# B&R Automation Studio project EFI (part 22)

#### OutputsP5.st
```iecst
ACTION OutputsP5:

(*CABINET 01*)

	//X20DOF322_009
	X20DOF322_009.DOutput[1]:=gBlockOutputs[1].xShotLine1;
	X20DOF322_009.DOutput[2]:=gBlockOutputs[1].xShotLine2;
	X20DOF322_009.DOutput[3]:=gBlockOutputs[1].xEnableDobleShot;
	X20DOF322_009.DOutput[4]:=gMachine.Out.xResetCB1;
	X20DOF322_009.DOutput[5]:=gMachine.Out.xResetRouter;
	X20DOF322_009.DOutput[6]:= FALSE;								//SPARE
	X20DOF322_009.DOutput[7]:=gMachine.Out.xAirSupply;
	X20DOF322_009.DOutput[8]:=gMachine.Out.xGreenLight;
	X20DOF322_009.DOutput[9]:=gMachine.Out.xLightReset;
	X20DOF322_009.DOutput[10]:=gMachine.Out.xBuzzerButtonPanel;
	X20DOF322_009.DOutput[11]:= TRUE;
	X20DOF322_009.DOutput[12]:= FALSE;								//SPARE
	X20DOF322_009.DOutput[13]:= FALSE;								//SPARE
	X20DOF322_009.DOutput[14]:= FALSE;								//SPARE
	X20DOF322_009.DOutput[15]:= FALSE;								//SPARE
	X20DOF322_009.DOutput[16]:= FALSE;								//SPARE

	// X20DOF322_010
	X20DOF322_010.DOutput[1]:= gInksOutputs[1].xOutPowPrintHead;
	X20DOF322_010.DOutput[2]:= gInksOutputs[2].xOutPowPrintHead;
	X20DOF322_010.DOutput[3]:= gInksOutputs[3].xOutPowPrintHead;
	X20DOF322_010.DOutput[4]:= gInksOutputs[4].xOutPowPrintHead;
	X20DOF322_010.DOutput[5]:= gInksOutputs[5].xOutPowPrintHead;
	X20DOF322_010.DOutput[6]:= gInksOutputs[6].xOutPowPrintHead;
	X20DOF322_010.DOutput[7]:= gInksOutputs[7].xOutPowPrintHead;
	X20DOF322_010.DOutput[8]:= gInksOutputs[8].xOutPowPrintHead;
	X20DOF322_010.DOutput[9]:= gInksOutputs[1].xOutBarResistance;
	X20DOF322_010.DOutput[10]:= gInksOutputs[2].xOutBarResistance;
	X20DOF322_010.DOutput[11]:= gInksOutputs[3].xOutBarResistance;
	X20DOF322_010.DOutput[12]:= gInksOutputs[4].xOutBarResistance;
	X20DOF322_010.DOutput[13]:= gInksOutputs[5].xOutBarResistance;
	X20DOF322_010.DOutput[14]:= gInksOutputs[6].xOutBarResistance;
	X20DOF322_010.DOutput[15]:= gInksOutputs[7].xOutBarResistance;
	X20DOF322_010.DOutput[16]:= gInksOutputs[8].xOutBarResistance;

	//X20DOF322_011
	X20DOF322_011.DOutput[1] := gInksOutputs[1].xSolenoid1;
	X20DOF322_011.DOutput[2] := gInksOutputs[2].xSolenoid1;
	X20DOF322_011.DOutput[3] := gInksOutputs[1].xSolenoid2;
	X20DOF322_011.DOutput[4] := gInksOutputs[2].xSolenoid2;
	X20DOF322_011.DOutput[5] := gInksOutputs[3].xSolenoid1;
	X20DOF322_011.DOutput[6] := gInksOutputs[4].xSolenoid1;
	X20DOF322_011.DOutput[7] := gInksOutputs[3].xSolenoid2;
	X20DOF322_011.DOutput[8] := gInksOutputs[4].xSolenoid2;
	X20DOF322_011.DOutput[9] := gInksOutputs[5].xSolenoid1;
	X20DOF322_011.DOutput[10] := gInksOutputs[6].xSolenoid1;
	X20DOF322_011.DOutput[11] := gInksOutputs[5].xSolenoid2;
	X20DOF322_011.DOutput[12] := gInksOutputs[6].xSolenoid2;
	X20DOF322_011.DOutput[13] := gInksOutputs[7].xSolenoid1;
	X20DOF322_011.DOutput[14] := gInksOutputs[8].xSolenoid1;
	X20DOF322_011.DOutput[15] := gInksOutputs[7].xSolenoid2;
	X20DOF322_011.DOutput[16] := gInksOutputs[8].xSolenoid2;

	//X20DOF322_012
	X20DOF322_012.DOutput[1]:=gInksOutputs[1].xReliefValve;
	X20DOF322_012.DOutput[2]:=gInksOutputs[2].xReliefValve;
	X20DOF322_012.DOutput[3]:=gInksOutputs[3].xReliefValve;
	X20DOF322_012.DOutput[4]:=gInksOutputs[4].xReliefValve;
	X20DOF322_012.DOutput[5]:=gInksOutputs[5].xReliefValve;
	X20DOF322_012.DOutput[6]:=gInksOutputs[6].xReliefValve;
	X20DOF322_012.DOutput[7]:=gInksOutputs[7].xReliefValve;
	X20DOF322_012.DOutput[8]:=gInksOutputs[8].xReliefValve;
	X20DOF322_012.DOutput[9]:= FALSE;								//SPARE
	X20DOF322_012.DOutput[10]:=FALSE;								//SPARE
	X20DOF322_012.DOutput[11]:=FALSE;								//SPARE
	X20DOF322_012.DOutput[12]:=FALSE;								//SPARE
	X20DOF322_012.DOutput[13]:=FALSE;								//SPARE
	X20DOF322_012.DOutput[14]:=FALSE;								//SPARE
	X20DOF322_012.DOutput[15]:=FALSE;								//SPARE
	X20DOF322_012.DOutput[16]:=FALSE;								//SPARE

	//X20DOF322_013
	X20DOF322_013.DOutput[1]:=gMachine.Out.xConsentL1;
	X20DOF322_013.DOutput[2]:=gMachine.Out.xConsentL2;
	X20DOF322_013.DOutput[3]:=gMachine.Out.xCompenserLine1;
	X20DOF322_013.DOutput[4]:=gMachine.Out.xCompenserLine2;
	X20DOF322_013.DOutput[5]:=gMachine.Out.xYellowLight;
	X20DOF322_013.DOutput[6]:=gMachine.Out.xRedLight;
	X20DOF322_013.DOutput[7]:=gMachine.Out.xLine1ReadyToClean;
	X20DOF322_013.DOutput[8]:=gMachine.Out.xLine2ReadyToClean;
	X20DOF322_013.DOutput[9]:=gMachine.Out.xSuctionTurbine;
	X20DOF322_013.DOutput[10]:= gJamDetect[1].Outputs.xJamTestSignal[1] OR gJamDetect[2].Outputs.xJamTestSignal[1];
	X20DOF322_013.DOutput[11]:=gJamDetect[1].Outputs.xJamTestSignal[2] OR gJamDetect[2].Outputs.xJamTestSignal[2];
	X20DOF322_013.DOutput[12]:=gJamDetect[1].Outputs.xJamTestSignal[3] OR gJamDetect[2].Outputs.xJamTestSignal[3];
	X20DOF322_013.DOutput[13]:=gJamDetect[1].Outputs.xJamTestSignal[4] OR gJamDetect[2].Outputs.xJamTestSignal[4];
	X20DOF322_013.DOutput[14]:= FALSE;								//SPARE
	X20DOF322_013.DOutput[15]:= FALSE;								//SPARE
	X20DOF322_013.DOutput[16]:= FALSE;								//SPARE

	// X20AO4622_017 	(*  BAR A *) 	(*  BAR B *)
	X20AO4622_017.AOutput[1]:= gInksOutputs[1].iDutyCycleNegative;
	X20AO4622_017.AOutput[2]:= gInksOutputs[2].iDutyCycleNegative;
	X20AO4622_017.AOutput[3]:= gInksOutputs[1].iDutyCycleFilling;
	X20AO4622_017.AOutput[4]:= gInksOutputs[2].iDutyCycleFilling;

	// X20AO4622_018 	(*  BAR C *) 	(*  BAR D *)
	X20AO4622_018.AOutput[1]:= gInksOutputs[3].iDutyCycleNegative;
	X20AO4622_018.AOutput[2]:= gInksOutputs[4].iDutyCycleNegative;
	X20AO4622_018.AOutput[3]:= gInksOutputs[3].iDutyCycleFilling;
	X20AO4622_018.AOutput[4]:= gInksOutputs[4].iDutyCycleFilling;

	// X20AO4622_019 	(*  BAR E *) 	(*  BAR F *)
	X20AO4622_019.AOutput[1]:= gInksOutputs[5].iDutyCycleNegative;
	X20AO4622_019.AOutput[2]:= gInksOutputs[6].iDutyCycleNegative;
	X20AO4622_019.AOutput[3]:= gInksOutputs[5].iDutyCycleFilling;
	X20AO4622_019.AOutput[4]:= gInksOutputs[6].iDutyCycleFilling;

	// X20AO4622_020 	(*  BAR G *) 	(*  BAR H *)
	X20AO4622_020.AOutput[1]:= gInksOutputs[7].iDutyCycleNegative;
	X20AO4622_020.AOutput[2]:= gInksOutputs[8].iDutyCycleNegative;
	X20AO4622_020.AOutput[3]:= gInksOutputs[7].iDutyCycleFilling;
	X20AO4622_020.AOutput[4]:= gInksOutputs[8].iDutyCycleFilling;

	// X20AO4622_100 THICKNESS SENSOR RESET
	X20AI2636_100.DOutput[1] := gDing.Out.xReset;;  // Reset the target fault

	// SI UNIT BK1
	SiUnitPwrLnkBK1.Output01_16.0 := gBlockOutputs[1].xTrayIn;
	SiUnitPwrLnkBK1.Output01_16.1 := gBlockOutputs[1].xTrayOut;
	SiUnitPwrLnkBK1.Output01_16.2 := gMachine.commands.CleanBelt.xCleanBeltPump;
	SiUnitPwrLnkBK1.Output01_16.3 := gBlockOutputs[1].xVenturi;
	SiUnitPwrLnkBK1.Output01_16.4 := gBlockOutputs[1].xCleaningWaterPump;
	SiUnitPwrLnkBK1.Output01_16.5 := gMachine.commands.CleanBelt.xPistonFlojet;
	SiUnitPwrLnkBK1.Output01_16.6 := FALSE;
	SiUnitPwrLnkBK1.Output01_16.7 := FALSE;
	SiUnitPwrLnkBK1.Output01_16.8 := FALSE;
	SiUnitPwrLnkBK1.Output01_16.9 := FALSE;
	SiUnitPwrLnkBK1.Output01_16.10 := FALSE;
	SiUnitPwrLnkBK1.Output01_16.11 := FALSE;
	SiUnitPwrLnkBK1.Output01_16.12 := FALSE;
	SiUnitPwrLnkBK1.Output01_16.13 := FALSE;
	SiUnitPwrLnkBK1.Output01_16.14 := FALSE;
	SiUnitPwrLnkBK1.Output01_16.15 := FALSE;

END_ACTION
```

#### OutputsShield.st
```iecst
ACTION OutputsShield:

	//X3 PLC
	X3.DOutput[1]:= FALSE;
	X3.DOutput[2]:= gMachine.Out.xPC2Start;
	X3.DOutput[3]:= gMachine.Out.xResetCB1;
	X3.DOutput[4]:= gMachine.Out.xResetRouter;

	// X20DOF322_005
	X20DOF322_005.DOutput[1]	:= gInksOutputs[1].xOutPowPrintHead;
	X20DOF322_005.DOutput[2]	:= gInksOutputs[2].xOutPowPrintHead;
	X20DOF322_005.DOutput[3]	:= gInksOutputs[1].xOutBarResistance;
	X20DOF322_005.DOutput[4]	:= gInksOutputs[2].xOutBarResistance;
	X20DOF322_005.DOutput[5]	:= gInksOutputs[1].xSolenoid1;
	X20DOF322_005.DOutput[6]	:= gInksOutputs[2].xSolenoid1;
	X20DOF322_005.DOutput[7]	:= gInksOutputs[1].xSolenoid2;
	X20DOF322_005.DOutput[8]	:= gInksOutputs[2].xSolenoid2;
	X20DOF322_005.DOutput[9]	:= gInksOutputs[1].xReliefValve;
	X20DOF322_005.DOutput[10]	:= gInksOutputs[2].xReliefValve;
	X20DOF322_005.DOutput[11]	:= FALSE;
	X20DOF322_005.DOutput[12]	:= gChiller[1].Out.xStart;
	X20DOF322_005.DOutput[13]	:= gMachine.Out.xCoolingPCStart;//Implement
	X20DOF322_005.DOutput[14]	:= gBlock[1].Out.xEnableDobleShot;
	X20DOF322_005.DOutput[15]	:= gBlock[1].Out.xShotLine1;
	X20DOF322_005.DOutput[16]	:= gBlock[1].Out.xShotLine2;

	// X20DOF322_006
	X20DOF322_006.DOutput[1]	:= gMachine.Out.xConsentL1;
	X20DOF322_006.DOutput[2]	:= gMachine.Out.xConsentL2;
	X20DOF322_006.DOutput[3]	:= gMachine.Out.xCompenserLine1;
	X20DOF322_006.DOutput[4]	:= gMachine.Out.xCompenserLine2;
	X20DOF322_006.DOutput[5]	:= gMachine.Out.xYellowLight;
	X20DOF322_006.DOutput[6]	:= gMachine.Out.xRedLight;
	X20DOF322_006.DOutput[7]	:= gMachine.Out.xLine1ReadyToClean;
	X20DOF322_006.DOutput[8]	:= gMachine.Out.xLine2ReadyToClean;
	X20DOF322_006.DOutput[9]	:= gMachine.Out.xSuctionTurbine;
	X20DOF322_006.DOutput[10]	:= FALSE;
	X20DOF322_006.DOutput[11]	:= FALSE;
	X20DOF322_006.DOutput[12]	:= TRUE;
	X20DOF322_006.DOutput[13]	:= gMachine.Out.xAirSupply;
	X20DOF322_006.DOutput[14]	:= gMachine.Out.xGreenLight;
	X20DOF322_006.DOutput[15]	:= gMachine.Out.xLightReset;
	X20DOF322_006.DOutput[16]	:= gMachine.Out.xBuzzerButtonPanel;

	// SI UNIT BK1
	SiUnitBK1.Output01_08.0		:= gBlockOutputs[1].xTrayIn;
	SiUnitBK1.Output01_08.1		:= gBlockOutputs[1].xTrayOut;
	SiUnitBK1.Output01_08.2		:= gMachine.commands.CleanBelt.xCleanBeltPump;
	SiUnitBK1.Output01_08.3		:= gBlockOutputs[1].xVenturi;
	SiUnitBK1.Output01_08.4		:= gMachine.commands.CleanBelt.xPistonFlojet;
	SiUnitBK1.Output01_08.5		:= gBlockOutputs[1].xCleaningWaterPump;

	// X20AO4622_009	 (*  BAR A *)	 (*  BAR B *)
	X20AO4622_009.AOutput[1]:= gInksOutputs[1].iDutyCycleNegative;
	X20AO4622_009.AOutput[2]:= gInksOutputs[2].iDutyCycleNegative;
	X20AO4622_009.AOutput[3]:= gInksOutputs[1].iDutyCycleFilling;
	X20AO4622_009.AOutput[4]:= gInksOutputs[2].iDutyCycleFilling;

END_ACTION
```

### Program Logical/Printer/Sim/SimMachine (IEC)

#### Main.st - Init, cyclic, exit code
```iecst
PROGRAM _INIT

	URLHost := '127.0.0.1';

	Initialization;

	//Call variables to avoid unusefull warnings
	// Simple modification
	GlobalIO;
	DeviceComms;
	Dryer;
	InkBox;
	Motion;

END_PROGRAM

PROGRAM _CYCLIC

	MachineModelCode;

	General;

	UPS;

	Tests;

	LogTests;

	//Definition of the machine at the end of the code
	IF simMachineTypeEnumCopy<>gSimMachine.Parameters.MachineType THEN
		simMachineType := DINT_TO_INT(gSimMachine.Parameters.MachineType);
		IF simMachineTypeEnumCopy <> SIM_MACHINE_REAL THEN
			xNeedToRestartCPU := TRUE;
		END_IF
	END_IF
	IF simMachineType<>simMachineTypeCopy THEN
		gSimMachine.Parameters.MachineType := simMachineType;
	END_IF

	simMachineTypeCopy := simMachineType;
	simMachineTypeEnumCopy := gSimMachine.Parameters.MachineType;

	//Restart CPU if needed. Done with timer to allow other programs to use the new model and save it before restart
	tonRestart.IN := xNeedToRestartCPU;
	tonRestart.PT := T#300ms;
	tonRestart();
	IF tonRestart.Q THEN
		statusReset := SYSreset(enable:= TRUE, mode:= 2);
	END_IF

END_PROGRAM

PROGRAM _EXIT
	gEventLogManager; //Just here to be able to watch this var
END_PROGRAM
```

#### GlobalVariables.st
```iecst
ACTION GlobalIO:
	X20CPUData; (*Map: P4&EBRO*)
	X1; (*Map: P4&EBRO*)
	X2; (*Map: P4&EBRO*)
	X3; (*Map: P4&EBRO*)
	X20DOF322_001; (*Map: P4*)
	X20DIF371_001; (*Map: EBRO&S1400*)
	X20DIF371_002; (*Map: P4&EBRO&S1400*)
	X20DIF371_003; (*Map: P4&EBRO$S1400*)
	X20DOF322_004; (*Map: P4*)
	X20DIF371_004; (*Map: EBRO*)
	X20DIF371_005; (*Map: S1400*)
	X20DIF371_006; (*Map: S1400*)
	X20AI2636_005; (*Map: P4*)
	X20DOF322_005; (*Map: EBRO*)
	X20SLX402_006; (*	X20SI2100_010; Map: P4*)
	X20DOF322_006; (*Map: EBRO*)
	X20AI4322_008; (*Map: EBRO*)
	X20AI4322_102; (*Map: InkBox*)
	X20AI4322_202; (*Map: InkBox*)
	X20AI4322_302; (*Map: InkBox*)
	X20AT2222_103; (*Map: InkBox*)
	X20AT2222_203; (*Map: InkBox*)
	X20AT2222_303; (*Map: InkBox*)
	X20DOF322_104; (*Map: InkBox*)
	X20DOF322_204; (*Map: InkBox*)
	X20DOF322_304; (*Map: InkBox*)
	X20AO4622_105; (*Map: InkBox*)
	X20AO4622_205; (*Map: InkBox*)
	X20AO4622_305; (*Map: InkBox*)
	X20DI9372_008; (*Map: S1400*)
	X20AO4622_009; (*Map: EBRO*)
	X20DOF322_009; (*Map:S1400*)
	X20DOF322_010; (*Map:S1400*)
	X20AT4222_010; (*Map: EBRO*)
	X20DOF322_011; (*Map:S1400*)
	X20DOF322_012; (*Map:S1400*)
	X20DOF322_013; (*Map:S1400*)
	X20AI8321_015; (*Map:S1400*)
	X20AI8321_016; (*Map:S1400*)
	X20AI8321_111; (*Map:S1400*)
	X20AI8321_112; (*Map:S1400*)
	X20AI8321_113; (*Map:S1400*)
	X20AI8321_018; (*Map:S1400*)
	X20AI8321_019; (*Map:S1400*)
	X20AO4622_017; (*Map:S1400*)
	X20AO4622_018; (*Map:S1400*)
	X20AO4622_019; (*Map:S1400*)
	X20AO4622_020; (*Map:S1400*)
	X20AT4222_022; (*Map:S1400*)
	X20AT4222_023; (*Map:S1400*)
	X20AI2636_024; (*Map:S1400*)
	X20AI8321_025;
	X20AI8321_024;
	X20DIF371_024; (*Map:S1400*)
	X20AI8321_026; (*Map:S1400*)
	X20AT4222_027;
	X20AT4222_028;
	X20AT4222_029; (*Map:S1400*)
	X20AT4222_030; (*Map:S1400*)
	X20DIF371_030; (*Map: P4*)
	X20AI2636_100;
	X20DIF371_101; (*Map: P4 & Map: InkBox*)
	X20DIF371_102; (*Map: P4*)
	X20DIF371_103; (*Map: P4*)
	X20DIF371_104; (*Map: P4*)
	X20DIF371_105; (*Map: P4*)
	X20DIF371_106; (*Map: P4*)
	X20DI9372_107; (*Map: P4*)
	X20DIF371_107; (*Map: P4*)
	X20DC4395_104; (*Map: P4*)
	X20DC4395_105; (*Map: P4*)
	X20DOF322_106; (*Map: P4*)
	X20DOF322_107; (*Map: P4*)
	X20DOF322_108; (*Map: P4*)
	X20DOF322_109; (*Map: P4*)
	X20DOF322_110; (*Map: P4*)
	X20AI8321_109; (*Map: P4*)
	X20AI8321_110; (*Map: P4*)
	X20AO4622_111; (*Map: P4*)
	X20AO4622_112; (*Map: P4*)
	X20AO4622_113; (*Map: P4*)
	X20AO4622_114; (*Map: P4*)
	X20AO4622_115; (*Map: P4*)
	X20AO4622_116; (*Map: P4*)
	X20AO4622_117; (*Map: P4*)
	X20AT4222_114; (*Map: P4*)
	X20AT4222_115; (*Map: P4*)
	X20AT4222_116; (*Map: P4*)
	X20AT4222_117; (*Map: P4*)
	X20AT4222_118; (*Map: P4*)
	X20AT4222_119; (*Map: P4*)
	X20AT4222_120; (*Map: P4*)
	X20AT4222_121; (*Map: P4*)
	X20CS1030_150; (*Map: P4*)
	X20CS1030_151; (*Map: P4*)
	X20PS3300_114; (*Map: P4*)
	X20PS3300_106; (*Map: P4*)
	X20PS3300_152; (*Map: P4*)
	X20DIF371_153; (*Map: P4*)
	X20DIF371_154; (*Map: P4*)
	X20DOF322_155; (*Map: P4*)
	X20AI8221_156; (*Map: P4*)
	X20AO4622_157; (*Map: P4*)
	X20AO4622_158; (*Map: P4*)
	X20SI8110_117; (*Map: P4*)
	X20SO2110_118; (*Map: P4*)
	X20DIF371_201; (*Map: P4 & InkBox*)
	X20DIF371_202; (*Map: P4*)
	X20DIF371_203; (*Map: P4*)
	X20DIF371_301; (*Map: InkBox*)
	X20DC4395_204; (*Map: P4*)
	X20DC4395_205; (*Map: P4*)
	X20DOF322_205; (*Map: Dryer*)
	X20DOF322_206; (*Map: P4*)
	X20DOF322_207; (*Map: P4*)
	X20DOF322_208; (*Map: P4*)
	X20AI8321_207; (*Map: P4*)
	X20AI8321_209; (*Map: P4*)
	X20AI8321_210; (*Map: P4*)
	X20AO4622_208; (*Map: Dryer*)
	X20AO4622_211; (*Map: P4*)
	X20AO4622_212; (*Map: P4*)
	X20AO4622_213; (*Map: P4*)
	X20AT4222_209; (*Map: Dryer*)
	X20AT4222_214; (*Map: P4*)
	X20AT4222_215; (*Map: P4*)
	X20AT4222_216; (*Map: P4*)
	X20SI8110_217; (*Map: P4*)
	X20SO2110_218; (*Map: P4*)
	Reserve01;
	SiUnitBK1;
	SiUnitBK2;
	SiUnitPwrLnkBK1;
	Pdc_X20DIF371_001;
	Pdc_X20DIF371_002;
	Pdc_X20DIF371_003;
	Pdc_X20DIF371_004;
	Pdc_X20DIF371_005;
	Pdc_X20DIF371_006;
	X20PS3300_007;
	Pdc_X20DIF371_020;
	Pdc_X20DIF371_021;
	X20PS3300_022;
	Pdc_X20DOF322_023;
	Pdc_X20DIF371_1;
	Pdc_X20DIF371_2;
	Pdc_X20DIF371_3;
	Pdc_X20DOF322_008;
	Pdc_X20DOF322_009;
	Pdc_X20DOF322_010;
	Pdc_X20DOF322_1;
	Pdc_X20DIF371_040;
	Pdc_X20DOF322_011;
	X20IF1072_SS1;
	X20SM1436_007;
	X20SM1436_008;
	X20SM1436_011;
	X20SM1436_012;
	X20SM1436_111;
	X20SM1436_112;
	X20PS3300_014;
	X20PS3300_021;
	X20BC0083;
	X20PS9400;
END_ACTION

ACTION DeviceComms:
	gIclaNetData;

	gReceivedDataModbTransport;
	gToWriteDataModbTransport;

END_ACTION

ACTION Dryer:

	gDryer;
	gDryerLocalData;
	gDryerRemoteData;
	gNirAdphos;
	gArcLampGew;
	gSimpleBlock;
	gIndexSimpleBlock;

	gPermanentArcLampGew;
	gPermanentNirAdphos;
	gPermanentDryer;
	gPermanentInkBox;
	gPermanentSimpleBlock;

	gSimArcLamp;
	gSimNirAdphos;
	gSimSimpleBlock;

END_ACTION

ACTION InkBox:

	gInkBox;

END_ACTION

ACTION Motion:

	gAxisStepper;

END_ACTION
```

#### SimMachine.var - Local variables
```iecst
VAR
	iIndexPsu : USINT;
	iSimIndex : USINT; (*Index for loops in simulation*)
	simEventLog : EventLog_typ;
	webClient : httpClient;
	ResponseHeader : httpResponseHeader_t;
	RequestData : STRING[3000];
	ResponseData : STRING[3000];
	URLHost : STRING[80];
	URIHost : STRING[80];
	xTestPrepareMachine : BOOL; (*This value must be used as active while pressed by the visualization*)
	xTestPrePrepare : BOOL; (*This value must be used as active while pressed by the visualization*)
	xTestBeltTests : BOOL; (*This value must be used as active while pressed by the visualization*)
	xTestConsents : BOOL; (*This value must be used as active while pressed by the visualization*)
	xTestBlock : BOOL; (*This value must be used as active while pressed by the visualization*)
	xTestTrVacuum : BOOL;
	xTestLine : BOOL; (*This value must be used as active while pressed by the visualization*)
	xTestCleaning : BOOL; (*This value must be used as active while pressed by the visualization*)
	testMonitor : UtMgrMonitor;
	ctrlBlock2 : UINT;
	simMachineType : INT;
	simMachineTypeCopy : INT;
	simMachineTypeEnumCopy : SimMachineType;
	xBlockExists2 : BOOL;
	statusReset : UINT;
	tonRestart : TON;
	xNeedToRestartCPU : BOOL;
	stEventLogTests : EventLog_typ;
END_VAR
```

### Program Logical/Printer/Sim/SimMachine_Fast (IEC)

#### Main.st - Init, cyclic, exit code
```iecst
PROGRAM _INIT

	InitialDataForMedia;
	PreparingMethodComms;

	InitialDataForMediaEnergy;
	PreparingMethodEnergyComms;

END_PROGRAM

PROGRAM _CYCLIC

	Media;

	// Sending information to the new boards
	Stack;
	StackEnergy;

END_PROGRAM
```

#### StackEnergy.st
```iecst
ACTION StackEnergy:

	(* UA_MethodCall - call methode *)
	InputArguments_Energy[0].Name := 'MediaData';
	InputArguments_Energy[0].Value := '::SimMachFst:NewMediaData_Energy';
	OutputArguments_Energy[0].Name := 'Result';
	OutputArguments_Energy[0].Value := '::SimMachFst:MethodResult_Energy';
	UA_MethodCall_Energy(Execute := ExecuteMethodCall_Energy,
		ConnectionHdl := ConnectionHdl_Energy,
		MethodHdl := MethodHdl_Energy,
		Timeout := T#10s,
		InputArguments := InputArguments_Energy,
		OutputArguments := OutputArguments_Energy);
	IF NOT UA_MethodCall_Energy.Busy THEN
		ExecuteMethodCall_Energy := FALSE;
		IF UA_MethodCall_Energy.Done THEN
			NewMediaData_Energy.MediaData.rLength := NewMediaData_Energy.MediaData.rLength + 1;
		END_IF
		IF UA_MethodCall_Energy.Error THEN
			NewMediaData_Energy.MediaData.rDocLength := NewMediaData_Energy.MediaData.rDocLength + 1;
		END_IF
	END_IF

	// Managing the automatic sending. Just Energy when enabled to Dry
	IF NOT gThicknessCtrl.status.xNewMediaStackEnabled OR NOT gThicknessCtrl.parameters.Dry.xDryStack THEN
		RETURN;
	END_IF

	IF (gSimMachine.Parameters.Stack.iMediaQuantityToKeepLoaded <= gThicknessCtrl.status.Stack.iNewMediaLoadedL1 + gThicknessCtrl.status.Stack.iNewMediaLoadedL2) THEN
		RETURN;
	END_IF

	// Adding a timer to avoid not working the method
	tonNotCallingMethod_Energy.IN := NOT UA_MethodCall_Energy.Busy;
	tonNotCallingMethod_Energy.PT := t#500ms;
	tonNotCallingMethod_Energy();
	IF EDGEPOS(tonNotCallingMethod_Energy.Q) THEN
		ExecuteMethodCall_Energy := TRUE;
	END_IF

END_ACTION

ACTION InitialDataForMediaEnergy:

	NewMediaData_Energy.MediaData.iLine := 1;
	NewMediaData_Energy.MediaData.xHasWhite := FALSE;
	NewMediaData_Energy.MediaData.rThickness := 3;
	NewMediaData_Energy.MediaData.rMargin := 2;
	NewMediaData_Energy.MediaData.rWidth := 1400;
	NewMediaData_Energy.MediaData.rLength := 1000;
	NewMediaData_Energy.MediaData.rCrossOffset := -700;
	NewMediaData_Energy.MediaData.rDocWidth := 1400;
	NewMediaData_Energy.MediaData.rDocLength := 950;
	NewMediaData_Energy.MediaData.rDocCrossOffset := -700;
	NewMediaData_Energy.MediaData.rDocProcessOffset := 0;

	//Just to see some data
	NewMediaData_Energy.Energy.iPower[0,0] := 50;
	NewMediaData_Energy.Energy.iPower[1,0] := 50;
	NewMediaData_Energy.Energy.iPower[0,1] := 50;

END_ACTION

ACTION PreparingMethodEnergyComms:

	ExecuteConnect_Energy := TRUE;

	(* UA_Connect - establish connection to OPC UA Server *)
	SessionConnectInfo_Energy.SecurityMsgMode := UASecurityMsgMode_None;
	SessionConnectInfo_Energy.SecurityPolicy := UASecurityPolicy_None;
	SessionConnectInfo_Energy.TransportProfile := UATP_UATcp;
	SessionConnectInfo_Energy.UserIdentityToken.UserIdentityTokenType := UAUITT_Username;
	SessionConnectInfo_Energy.UserIdentityToken.TokenParam1 := 'PressCore';
	SessionConnectInfo_Energy.UserIdentityToken.TokenParam2 := 'h98o76';
	SessionConnectInfo_Energy.SessionTimeout := T#1m;
	SessionConnectInfo_Energy.MonitorConnection := T#10s;

	UA_Connect_Energy(Execute := ExecuteConnect_Energy,
		ServerEndpointUrl := 'opc.tcp://localhost:4840',
		SessionConnectInfo := SessionConnectInfo_Energy,
		Timeout := T#10s);
	IF NOT UA_Connect_Energy.Busy THEN
		ExecuteConnect_Energy := FALSE;
		IF UA_Connect_Energy.Done THEN
			ConnectionHdl_Energy := UA_Connect_Energy.ConnectionHdl;
			////// NEXT
			ExecuteGetnamespaceindex_Energy := TRUE;
		END_IF
		IF UA_Connect_Energy.Error THEN
			ConnectionHdl_Energy := 0;
		END_IF
	END_IF

	(* UA_GetNamespaceIndex - read index of required namespace for PVs *)
	UA_GetNamespaceIndex_Energy(Execute := ExecuteGetnamespaceindex_Energy,
		ConnectionHdl := ConnectionHdl_Energy,
		NamespaceUri := 'http://br-automation.com/OpcUa/PLC/PV/',
	Timeout := T#5s);
	IF NOT UA_GetNamespaceIndex_Energy.Busy THEN
		ExecuteGetnamespaceindex_Energy := FALSE;
		IF UA_GetNamespaceIndex_Energy.Done THEN
			NamespaceIndex_Energy := UA_GetNamespaceIndex_Energy.NamespaceIndex;
			////// NEXT
			ExecuteMethodGetHandle_Energy := TRUE;
		END_IF
		IF UA_GetNamespaceIndex_Energy.Error THEN
			NamespaceIndex_Energy := 0;
		END_IF
	END_IF

	(* UA_MethodGetHandle - get a handle for required methode *)
	ObjectNodeID_Energy.NamespaceIndex := NamespaceIndex_Energy;
	ObjectNodeID_Energy.Identifier := '::ThickPos';
	ObjectNodeID_Energy.IdentifierType := UAIdentifierType_String;
	MethodNodeID_Energy.NamespaceIndex := NamespaceIndex_Energy;
	MethodNodeID_Energy.Identifier := '::ThickPos:LoadNewMediaEnergy';
	MethodNodeID_Energy.IdentifierType := UAIdentifierType_String;
	UA_MethodGetHandle_Energy(Execute := ExecuteMethodGetHandle_Energy,
		ConnectionHdl := ConnectionHdl_Energy,
		ObjectNodeID := ObjectNodeID_Energy,
		MethodNodeID := MethodNodeID_Energy,
		Timeout := T#10s);
	IF NOT UA_MethodGetHandle_Energy.Busy THEN
		ExecuteMethodGetHandle_Energy := FALSE;
		IF UA_MethodGetHandle_Energy.Done THEN
			MethodHdl_Energy := UA_MethodGetHandle_Energy.MethodHdl;
			////// NEXT
			// READY TO COMMUNICATE
		END_IF
		IF UA_MethodGetHandle_Energy.Error THEN
			MethodHdl_Energy := 0;
		END_IF
	END_IF

END_ACTION
```

- Visualisation Logical/Printer/Sim/SimVisu (not shown)

### Program Logical/Printer/Sim/TestResources (IEC)

#### TestResources.st - Init, cyclic, exit code
```iecst
PROGRAM _CYCLIC

	rVal := 0.6; //Complex value. Just a starting value
	FOR iIndex:=0 TO iMax DO
		rVal := rVal * SQRT(rVal);
	END_FOR;

END_PROGRAM
```

- Remote&LocalParams.graphml (not shown)

### Package Logical/Dryer/Config - Machine configurator

### Program Logical/Dryer/Config/Initialize (IEC) - Initialize program

#### Initialize.var
```iecst
VAR
	HWInfoCpu : HWInfo;
	projectInfo : ArProjectGetInfo;
END_VAR
```

### Program Logical/Dryer/Config/MachineConfigurator (IEC) - Machine configurator

#### MachineModel.st - Constant values according machine model
```iecst
ACTION MachineModel:

	//Assignation of machine model just when unnasigned
	IF gDryer.In.iMachineModelCode=0 THEN
		InputsMachineModel;
	END_IF

	// MachineModelAssignation
	// From the inputs of the type of machine readed by the inputs to the Parameter of the particular Type of Machine
	CASE gDryer.Pt.ConfigNameID OF

		GC_CONFIG_DRYER_NOZ2_ID:
			CASE gDryer.In.iMachineModelCode OF
				03: //Dryer Nozomi 2	|| 01-> 0000 0011
					gDryer.Pt.MachineModel:=DryerType_NOZ2_NIR_ARCLAMP;
				02: //Dryer Nozomi 2	|| 01-> 0000 0010
					gDryer.Pt.MachineModel:=DryerType_NOZ2_NIR;
				ELSE
					gDryer.Pt.MachineModel:=DryerNoType;

			END_CASE;

		GC_CONFIG_SIMDRYER_NOZ2_ID:
			CASE gDryer.In.iMachineModelCode OF
				03: // Nozomi2 Dryer		|| 01-> 0000 0011
					gDryer.Pt.MachineModel:= DryerType_NOZ2_NIR_ARCLAMP;
				02: // Nozomi2 Dryer		|| 01-> 0000 0010
					gDryer.Pt.MachineModel:= DryerType_NOZ2_NIR;

				ELSE
					gDryer.Pt.MachineModel:=DryerNoType;

			END_CASE;
			xChangedSimMachine := simMachine_copy <> gSimMachine.Parameters.MachineType;
			simMachine_copy := gSimMachine.Parameters.MachineType;

		ELSE
			gDryer.Pt.MachineModel:=DryerNoType;

	END_CASE

	//Assignation of the axis
	AxisAssignation;

	// Code To Kernel	(Tranfer the other codes)
	CASE gDryer.Pt.MachineModel OF
		DryerType_NOZ2_NIR_ARCLAMP:
			gDryer.St.iMachineModelCodeSW:=5001;

		DryerType_NOZ2_NIR:
			gDryer.St.iMachineModelCodeSW:=5002;

		ELSE
			gDryer.St.iMachineModelCodeSW:= 0;

	END_CASE;

END_ACTION

ACTION InputsMachineModel:

	CASE gDryer.Pt.ConfigNameID OF

		GC_CONFIG_DRYER_NOZ2_ID:
			gDryer.In.iMachineModelCode.3:= X20DIF371_201.DInput[16];
			gDryer.In.iMachineModelCode.2:= X20DIF371_201.DInput[15];
			gDryer.In.iMachineModelCode.1:= X20DIF371_201.DInput[14];
			gDryer.In.iMachineModelCode.0:= X20DIF371_201.DInput[13];

	END_CASE;

END_ACTION

ACTION AxisAssignation:

	IF gDryer.Pt.ConfigNameID = GC_CONFIG_SIMDRYER_NOZ2_ID THEN
		Axis_Simulation;
		RETURN;
	END_IF

	//Name of the Axis as defined in Hardware
	CASE gDryer.Pt.MachineModel OF

		DryerType_NOZ2_NIR,
		DryerType_NOZ2_NIR_ARCLAMP:
			Axis_DryerNoz2;

		ELSE
			//No machine assigned
			RETURN;

	END_CASE

END_ACTION

ACTION Axis_Simulation:

	(* Insert code here *)
    //Name of the Axis as defined in Hardware
	gAxis[1].Parameter.Init.AxisObjectName			:=	'gAxis01';	//Instance_Belt
	gAxis[2].Parameter.Init.AxisObjectName			:=	'gAxis02';	//Instance_BK1

	gAxisInverter[1].Parameters.Hardware.PowerLinkInterface := 'IF3';
	gAxisInverter[1].Parameters.Hardware.Node := 81;
	gAxisInverter[1].Parameters.AccelerationTime := 1;
	gAxisInverter[1].Parameters.DecelerationTime := 1;
	gAxisInverter[1].Parameters.CommsType := COMMS_POWERLINK;
	gAxisInverter[2].Parameters.Hardware.PowerLinkInterface := 'IF3';
	gAxisInverter[2].Parameters.Hardware.Node := 82;
	gAxisInverter[2].Parameters.AccelerationTime := 1;
	gAxisInverter[2].Parameters.DecelerationTime := 1;
	gAxisInverter[2].Parameters.CommsType := COMMS_POWERLINK;

	LoadDefaultServoConfig(ADR(gAxis[1]));
	LoadDefaultServoConfig(ADR(gAxis[2]));

END_ACTION

ACTION Axis_DryerNoz2:

	(* Insert code here *)
    //Name of the Axis as defined in Hardware
	gAxis[1].Parameter.Init.AxisObjectName			:=	'gAxis01';	//Instance_Belt
	gAxis[2].Parameter.Init.AxisObjectName			:=	'gAxis02';	//Instance_BK1

	// To choose communication protocol for VSDs while are UNDEFINED
	IF gAxisInverter[1].Parameters.CommsType = COMMS_UNDEFINED AND gAxisInverter[2].Parameters.CommsType = COMMS_UNDEFINED THEN
		IF gInverterSignalsPowerLink[1].In.ModuleOk AND gInverterSignalsPowerLink[2].In.ModuleOk THEN
			gAxisInverter[1].Parameters.CommsType := COMMS_POWERLINK;
			gAxisInverter[2].Parameters.CommsType := COMMS_POWERLINK;
		ELSIF gInverterSignalsCanOpen[1].In.ModuleOk AND gInverterSignalsCanOpen[2].In.ModuleOk THEN
			gAxisInverter[1].Parameters.CommsType := COMMS_CANOPEN;
			gAxisInverter[2].Parameters.CommsType := COMMS_CANOPEN;
		END_IF
	END_IF
	IF gAxisInverter[1].Parameters.CommsType = COMMS_POWERLINK THEN
		gAxisInverter[1].Parameters.Hardware.PowerLinkInterface := 'IF3';
		gAxisInverter[1].Parameters.Hardware.Node := 81;
		gAxisInverter[1].Parameters.AccelerationTime := 1;
		gAxisInverter[2].Parameters.Hardware.PowerLinkInterface := 'IF3';
		gAxisInverter[2].Parameters.Hardware.Node := 82;
		gAxisInverter[2].Parameters.DecelerationTime := 1;
	ELSIF gAxisInverter[1].Parameters.CommsType = COMMS_CANOPEN THEN
		gAxisInverter[1].Parameters.Hardware.Node := 81;
		gAxisInverter[1].Parameters.AccelerationTime := 1;
		gAxisInverter[1].Parameters.Hardware.PowerLinkInterface := 'IF7';
		gAxisInverter[2].Parameters.Hardware.Node := 82;
		gAxisInverter[2].Parameters.Hardware.PowerLinkInterface := 'IF7';
		gAxisInverter[2].Parameters.AccelerationTime := 1;
	END_IF

	LoadDefaultServoConfig(ADR(gAxis[1]));
	LoadDefaultServoConfig(ADR(gAxis[2]));

END_ACTION
```

#### MachineConfigurator.var - Local variables
```iecst
VAR
	iBlockIndex : USINT;
	DryerModelCopy : DryerModel_enum;
	xChangedSimMachine : BOOL;
	simMachine_copy : SimMachineType;
	iIndexBlock : USINT; (*Block Index to use a FOR*)
	iIndexTrVacc : USINT; (*TransportVacuum Index to use a FOR*)
END_VAR
```

- Program Logical/Dryer/Config/SavePermanent (IEC) (no source held here)

### HMI.var
```iecst
VAR
	AlarmsHistory : MpAlarmXHistory;
	AlarmsCore : MpAlarmXCore;
	xTest : BOOL;
	myValue : UDINT;
	xNone : BOOL;
	xActive : BOOL;
	xInactive : BOOL;
	xAck : BOOL;
	xUnAck : BOOL;
	myValue2 : DINT;
	myValueAck : DINT;
	xTest2 : BOOL;
	myValueAck2 : DINT;
	xSimulateMedia : BOOL;
	tonSimMedia : TON;
END_VAR
```

### Package Logical/Dryer/DryerCtrl - Controller commads to printer

- MachineStates.graphml (not shown)

### ReadmeMachineCtrl.txt
```
	(* From efi Cretaprint Almazora Castellon

	Machine Control is a manager of printers and based on two cyclic tasks.
	At first step, we have implemented on this case a slow cyclic task for belt cleaning, block cleaning, instant print shots, CB&Router resets, light beacon, buzzer sounds.
	All of them, are implemented using sequancial actions considered by main task named Machine_Ctrl_Slow.
	An important point is showed in GeneralMachineData.st
	It is an action where are all implemented all data that printer needs to be configured as logical for printing, from now on all parameters have to be paremeters defined by printer

	At the second part is Machine_Ctrl_Fast.st
	Machine_Ctrl_Fast cyclic task has more priority than Machine_Ctrl_Slow
	In thi cyclic task, we have to implement status of the printer, ie, Machine status: PRINTING, CLEANING, CAP... Also Alarms, orders, status, Heigh Detection

	*)
```

### Program Logical/Dryer/DryerCtrl/DryerCtrl_Fast (IEC)

#### DryerInputs.st - Operation/Mode active
```iecst
ACTION MachineInputs:

	ProductDetectSignals;

	//Probe -200C +500C. Range 700C
	gDryer.St.Temp.rBelt := ((INT_TO_REAL(gDryer.In.Temp.iBeltRaw)* 520.0)/32767.0)-20.0;
	gDryer.St.Temp.rBoardIn := ((INT_TO_REAL(gDryer.In.Temp.iBoardInRaw)* 520.0)/32767.0)-20.0;
	gDryer.St.Temp.rBoardOut := ((INT_TO_REAL(gDryer.In.Temp.iBoardOutRaw)* 520.0)/32767.0)-20.0;

	gDryer.St.Temp.rAirBlowerInput := ((INT_TO_REAL(gDryer.In.Temp.iAirBlowerInputRaw)* 250.0)/32767.0)-50.0;
	gDryer.St.Temp.rAirBlowerOutput := ((INT_TO_REAL(gDryer.In.Temp.iAirBlowerOutputRaw)* 250.0)/32767.0)-50.0;

END_ACTION

ACTION ProductDetectSignals:

	IF gDryer.In.ProductDetect.pPDSignalSensorL1 = 0 OR gDryer.In.ProductDetect.pPDSignalSensorL2 = 0 THEN
		RETURN;
	END_IF

	//Aggregated signals in the machine to clarify reading code
	xPDCarriageSignalL1 ACCESS gDryer.In.ProductDetect.pPDSignalSensorL1;
	xPDCarriageSignalL2 ACCESS gDryer.In.ProductDetect.pPDSignalSensorL2;

	gDryer.St.xProductDetectL1 := xPDCarriageSignalL1;
	gDryer.St.xProductDetectL2 := xPDCarriageSignalL2;

	gDryer.St.xAnyProductDetect := gDryer.St.xProductDetectL1 OR gDryer.St.xProductDetectL2;

	gDryer.St.xMediaDetected := gBasicDetectMedia.Status.xMediaPresent;

END_ACTION
```

#### MachineStates.st - Operation/Mode active
```iecst
ACTION MachineStates:

	// Mute	conditions
	// Impovement in Test:"xRestartAfterPCPLCError": This condition is necessary to remove souns when comnns are restablished

	gDryer.AutoCmd.xStart := EDGEPOS (tonStartButton.Q OR gDryer.In.Sw.xStart_GI);

	tonStop.IN := gDryer.In.Buttons.xStop OR gDryer.In.Sw.xStop_GI;
	tonStop.PT := T#2s;
	tonStop();
	gDryer.AutoCmd.xStop := (tonStop.Q OR EDGEPOS (gDryer.In.Buttons.xStop OR gDryer.In.Sw.xStop_GI)) AND NOT gDryer.St.AutoLocation.xRemote;
	gDryer.AutoCmd.xReset:= gDryer.In.Buttons.xReset OR gDryer.In.Sw.xReset_GI;

	gDryer.AutoCmd.xMuteAlarms:= gDryer.In.Sw.xMute_GI OR gDryer.In.xMute OR gDryer.AutoCmd.xReset;

	(* Manual/Auto/Zero *)

	// Automatic Mode
	iReasonNotEnterAuto.0 := gDryer.AlSummary.xAlarmCritical;
	//iReasonNotEnterAuto.1 := gDryer.Al.Warning.xFrontDoorOpened;
	//iReasonNotEnterAuto.2 := gDryer.Al.Warning.xRearDoorOpened;
	iReasonNotEnterAuto.3 := gSimpleBlock[1].Al.xAlrBarMtrNoRef AND gArcLampGew.Status.xInstalled; //Just not allow entering in auto if ArcLamp is installed
	gDryer.St.xNotAutoPossible := iReasonNotEnterAuto > 0;
	IF gDryer.In.Buttons.xAuto AND gDryer.In.Buttons.xReset AND iReasonNotEnterAuto = 0 THEN
		enPrinterState:=PRINTERGEN_AUTO;
	END_IF

	// Manual Mode
	IF gDryer.In.Buttons.xManual AND gDryer.In.Buttons.xReset THEN
		enPrinterState:=PRINTERGEN_MANUAL;
	END_IF

	// Zero Mode
	iReasonOut.0 := gDryer.In.Buttons.xZero;
	iReasonOut.1 := NOT gDryer.In.Buttons.xAuto AND enPrinterState=PRINTERGEN_AUTO; // It avoids manual state when safety is NOT ready
	iReasonOut.2 := NOT gDryer.In.Buttons.xManual AND enPrinterState=PRINTERGEN_MANUAL; // It avoids manual state when safety is NOT ready
	iReasonOut.3 := gDryer.AlSummary.xAlarmCritical AND enPrinterState=PRINTERGEN_AUTO;
	iReasonOut.4 := gDryer.Al.xAlrSafetySystemEStop;
	IF iReasonOut > 0	THEN
		IF enPrinterState<>PRINTERGEN_ZERO THEN
			LogOutOfAuto;
		END_IF
		enPrinterState:=PRINTERGEN_ZERO;
	END_IF

	//MachineStates
	gDryer.St.Mode.xZero	:= enPrinterState = PRINTERGEN_ZERO;
	gDryer.St.Mode.xManual	:= enPrinterState = PRINTERGEN_MANUAL;
	gDryer.St.Mode.xAuto	:= enPrinterState = PRINTERGEN_AUTO;
	// Updated state MANUAL, ZERO OR AUTO
	// This state is used on block, gbelt
	gDryer.St.StateMode:=enPrinterState;

	rsRunBeltOrderManual.SET   := gDryer.AutoCmd.xStart;
	rsRunBeltOrderManual.RESET1:= 	gDryer.St.AutoMode.xPause OR
									gDryer.AutoCmd.xStop OR
									gDryer.Al.xAlrSafetySystemEStop OR
									gDryer.Al.Alarm.xAlrJam OR
									NOT gDryer.St.Mode.xManual OR
									gDryer.Al.Alarm.xAlarmMountedMedia;

	rsRunBeltOrderManual();
	g_xRunBeltOrderManual:=rsRunBeltOrderManual.Q1;

	CASE enPrinterState OF

		PRINTERGEN_ZERO:
			WhileNotInAuto;

		PRINTERGEN_MANUAL:
			WhileNotInAuto;

		PRINTERGEN_AUTO:

			//Restore previous status
			IF gDryer.AutoCmd.iAutoMode=AUTO_NOT_VALID THEN
				gDryer.St.LocationControl := AutoLocationPrevious;
			END_IF

			IF EDGEPOS(gDryer.commands.xToLocal) THEN
				gDryer.commands.xToLocal:=FALSE;
				gDryer.St.LocationControl := MACHLOC_LOCAL;
			ELSIF EDGEPOS(gDryer.commands.xToRemote) THEN
				gDryer.commands.xToRemote:=FALSE;
				gDryer.St.LocationControl := MACHLOC_REMOTE;
			END_IF

			// Normal Cmd
			IF NOT gDryer.AlSummary.xAlarmStop AND NOT gDryer.Al.xAlrDisableGoToProduction AND
				// In lab mode doesnt go to production,is just starting belt
				( (gDryer.AutoCmd.xStart AND gDryer.AutoCmd.iAutoMode<>AUTO_BYPASS) OR gDryer.In.Sw.xToNormal_GI OR gDryer.St.AutoLocation.xRemote) THEN

				gDryer.AutoCmd.iAutoMode:=AUTO_PRODUCTION;
			END_IF

			//BYPASS
			IF gDryer.In.Sw.xToByPass_GI OR
				(EDGENEG(gDryer.In.xStart) AND NOT tonStartButton.Q AND (gDryer.AutoCmd.iAutoMode=AUTO_STOP) ) THEN

				gDryer.AutoCmd.iAutoMode:=AUTO_BYPASS;
			END_IF

			// STOP
			iReasonStop.0 := gDryer.AutoCmd.xStop;
			iReasonStop.1 := gDryer.AutoCmd.iAutoMode=AUTO_NOT_VALID;
			iReasonStop.2 := gDryer.AutoCmd.iAutoMode<>AUTO_BYPASS AND gDryer.AlSummary.xAlarmStop;
			IF iReasonStop > 0 THEN
				//Register last reason to Stop
				IF (gDryer.AutoCmd.iAutoMode<>AUTO_STOP) THEN iLastReasonStop := iReasonStop; END_IF
				gDryer.AutoCmd.iAutoMode:=AUTO_STOP;
			END_IF

	END_CASE

	//Define the individual bits for each state
	gDryer.St.AutoMode.xProduction	:= gDryer.AutoCmd.iAutoMode = AUTO_PRODUCTION;
	gDryer.St.AutoMode.xBypass		:= gDryer.AutoCmd.iAutoMode = AUTO_BYPASS;
	//gDryer.St.AutoMode.xLaboratory	:= gDryer.AutoCmd.iAutoMode = AUTO_LABORATORY;
	gDryer.St.AutoMode.xStop			:= gDryer.AutoCmd.iAutoMode = AUTO_STOP;
	gDryer.St.AutoMode.xProdORLab 	:= gDryer.St.AutoMode.xProduction OR gDryer.St.AutoMode.xLaboratory;
	gDryer.St.AutoMode.xProdORByPass 	:= gDryer.St.AutoMode.xProduction OR gDryer.St.AutoMode.xBypass;

	// State: Pause
	iReasonSetPause.0 := gDryer.In.Sw.xPause_GI;
	iReasonSetPause.1 := EDGEPOS(gDryer.St.AutoMode.xLaboratory);
	iReasonSetPause.2 := EDGEPOS(gDryer.St.Mode.xAuto) ;
	iReasonSetPause.3 := (EDGEPOS(gDryer.In.xStart) AND gBelt.states.xRuningBelt);
	srPauseMachine.SET:= iReasonSetPause > 0;

	iReasonResetPause.0 := EDGEPOS(gDryer.St.AutoMode.xBypass);
	iReasonResetPause.1 := EDGEPOS(gDryer.St.AutoMode.xProduction);
	iReasonResetPause.2 := gDryer.AutoCmd.xStart;
	iReasonResetPause.3 := (gDryer.St.AutoMode.xPause AND EDGEPOS(gDryer.In.xStart));
	iReasonResetPause.4 := gDryer.St.Mode.xZero;
	iReasonResetPause.5 := gDryer.St.AutoMode.xStop;
	srPauseMachine.RESET1:= iReasonResetPause > 0;

	srPauseMachine();
	gDryer.St.AutoMode.xPause := srPauseMachine.Q1;

	//Machine state to SW, is it used on SW? Or iBlockState?
	CASE gDryer.AutoCmd.iAutoMode OF
		AUTO_PRODUCTION:     gDryer.St.iAutoModeSW:= 1;
		AUTO_BYPASS:         gDryer.St.iAutoModeSW:= 2;
		AUTO_LABORATORY:     gDryer.St.iAutoModeSW:= 3;
		AUTO_STOP:           gDryer.St.iAutoModeSW:= 0;
	END_CASE

	tonStartButton(IN:= gDryer.In.xStart, PT:= T#1s);

	ton_ZeroMode(IN:= gDryer.St.Mode.xZero, PT:= T#100ms);

	gDryer.St.AutoLocation.xLocal := gDryer.St.LocationControl = MACHLOC_LOCAL;
	gDryer.St.AutoLocation.xLocalORManual := gDryer.St.LocationControl <> MACHLOC_REMOTE;
	gDryer.St.AutoLocation.xRemote := gDryer.St.LocationControl = MACHLOC_REMOTE;

	IF gDryer.St.AutoLocation.xRemote THEN
		DryerParams ACCESS ADR(gDryerRemoteData.Parameters);
		DryerSignalsAuto ACCESS ADR(gDryerRemoteData);
	ELSE
		DryerParams ACCESS ADR(gDryerLocalParams);
		DryerSignalsAuto ACCESS ADR(gDryerLocalSignals);
	END_IF

	IF EDGE(gDryer.St.AutoLocation.xRemote) THEN
		gDryerLocalSignals := gDryerLocalSignalsReseted;
		StoredParamsToWork;
	END_IF

	IF gDryer.St.AutoLocation.xRemote THEN
		StoredParamsToWork;
	ELSE
		WorkParamsToStored;
	END_IF

	//Assign to remote data local parameters without Sw interface
	gDryerRemoteData.Parameters.Media.rMargin := gDryerLocalParams.Media.rMargin;
	gDryerRemoteData.Parameters.Safety.rMaxBeltSpeedSetPoint := gDryerLocalParams.Safety.rMaxBeltSpeedSetPoint;

END_ACTION

ACTION WhileNotInAuto:

	//Store the first time previous Auto Location
	IF gDryer.AutoCmd.iAutoMode<>AUTO_NOT_VALID THEN
		AutoLocationPrevious := gDryer.St.LocationControl;
		gDryer.St.LocationControl := AutoLocationReseted;
	END_IF

	gDryer.AutoCmd.iAutoMode:=AUTO_NOT_VALID;

END_ACTION

ACTION StoredParamsToWork:
	gDryer.Pt.SW := DryerParams;
END_ACTION

ACTION WorkParamsToStored:
	DryerParams := gDryer.Pt.SW;
END_ACTION
```

#### ResetAlarms.st - Reset alarms
```iecst
ACTION ResetAlarms:

	gDryer.Al := stDryerAlarmsReseted;

END_ACTION
```

### Program Logical/Dryer/DryerCtrl/DryerCtrl_Slow (IEC)

#### DryerCtrl_Slow.st - Calling program actions
```iecst
PROGRAM _INIT

	versionPLC;

	PLC_Init(ADR(gPLC));

END_PROGRAM

PROGRAM _CYCLIC

	InternalPLC;

	VarsVersion;

	GeneralMachineData;

	// It allows CleanBelt action integrated on BeltManager
	CleanBelt;

	//Doors;

	// It allows to have consent lone in belt orders
	//[RGP] Execute "ConsentsLine" always. It was previously called if "gBelt.parameters.xExistConsentLine" was active and always was
	ConsentsLine;

	SuctionBlower;
	ResetRouterAndHub;

	AlarmsSlow;

	// Slow orders sent to the elements
	OrdersSlow;

	SoundBeacon;
	LightBeacon;

	gDryer.St.xStarted := TRUE;
	gDryer.St.exec.slow := gDryer.St.exec.slow +1;

END_PROGRAM
```

#### InternalPLC.st - Internal PLC Vars
```iecst
ACTION versionPLC:

    // Version
	gPLC.iVersion0:= 1;
	gPLC.iVersion1:= 67;	// Refactoring
	gPLC.iVersion2:= 394; 	// Updated ExtPack
	gPLC.iVersion3:= 187;

END_ACTION

ACTION InternalPLC:

	// PLC VARS
	IF gPLC.diCycleTime =0 THEN
		RTInfo_0(enable := TRUE);
		gPLC.diCycleTime:=RTInfo_0.cycle_time;  // Is a fix cycle time
		gPLC.xFirst_Scan:= RTInfo_0.init_reason=-1 OR RTInfo_0.init_reason=1 OR RTInfo_0.init_reason=2 OR RTInfo_0.init_reason=3;
		gPLC.xColdRestart:= RTInfo_0.init_reason=1;
		gPLC.xWarmRestart:= RTInfo_0.init_reason=2;
		gPLC.xDownloadRestart:= RTInfo_0.init_reason=3;

	ELSIF gPLC.xFirst_Scan THEN
		gPLC.xFirst_Scan:= FALSE;
		gPLC.xColdRestart:= FALSE;
		gPLC.xWarmRestart:= FALSE;
		gPLC.xDownloadRestart:= FALSE;
	END_IF

	//BLINK
	Blink_100ms.T_Blink:=T#100MS;
	Blink_100ms();
	gPLC.xBlk_100ms:= Blink_100ms.Out;

	Blink_200ms.T_Blink:=T#200MS;
	Blink_200ms();
	gPLC.xBlk_200ms:= Blink_200ms.Out;

	Blink_500ms.T_Blink:=T#500MS;
	Blink_500ms();
	gPLC.xBlk_500ms:= Blink_500ms.Out;

	Blink_1s.T_Blink:=T#1S;
	Blink_1s();
	gPLC.xBlk_1s:= Blink_1s.Out;

	Blink_2s.T_Blink:=T#2S;
	Blink_2s();
	gPLC.xBlk_2s:= Blink_2s.Out;

	Blink_5s.T_Blink:=T#5S;
	Blink_5s();
	gPLC.xBlk_5s:= Blink_5s.Out;

	// License counter	and  Keep alive
	IF EDGEPOS(gPLC.xBlk_1s) THEN
		gDryer.St.uiLicenseCounter:= gDryer.St.uiLicenseCounter+1;
	END_IF;

	//Setting Serial Name of the PLC
	setSerialNumber;

END_ACTION

ACTION setSerialNumber:

    // If the PLC has version, return
	IF brsstrlen(ADR(gDryer.St.HwData.SerialNumber)) > 0 THEN
		RETURN;
	END_IF

	IF EDGEPOS(gDryer.commands.SerialNumber.xExecute) THEN
		brsstrcpy(ADR(gDryer.St.HwData.SerialNumber),ADR(gDryer.commands.SerialNumber.SerialNumber));
		gDryer.commands.SerialNumber.xExecute := FALSE;
	END_IF

END_ACTION
```

#### VarsVersion.st
```iecst
// THIS CODE IS AUTOGENERATED. DO NOT MODIFY IT WITH AUTOMATION STUDIO
// Generation: 27/05/24 15:29:30
// Program version: 2.1.3.0

ACTION VarsVersion:

	gPLC.iVarsVersion0 := 1;
	gPLC.iVarsVersion1 := 3;
	gPLC.iVarsVersion2 := 1;
	gPLC.iVarsVersion3 := 41;

END_ACTION
```

#### Doors.st
```iecst
ACTION Doors:

	// AND REASONS
	iReasonReleaseDoors.0 := gDryer.St.Mode.xZero;
	iReasonReleaseDoors.1 := gNirAdphos.Status.rSurfaceTempModule[1] < 40 OR gDryer.In.xOpenDoorsKey;
	iReasonReleaseDoors.2 := gNirAdphos.Status.rSurfaceTempModule[2] < 40 OR gDryer.In.xOpenDoorsKey;
	xReleaseDoors := iReasonReleaseDoors >= 2#00111;

	// AND REASONS
	iReasonLockDoors.0 := gDryer.St.Mode.xAuto;
	xLockDoors := iReasonLockDoors >= 2#00001;

	IF xReleaseDoors (*AND gDryer.commands.xUnlockDoors*) THEN
		gDryer.Out.xLockFrontDoor := FALSE;
		gDryer.Out.xLockRearDoor := FALSE;
	END_IF

	IF xLockDoors THEN
		gDryer.Out.xLockFrontDoor := TRUE;
		gDryer.Out.xLockRearDoor := TRUE;
	END_IF

	//Just as an edge command
	gDryer.commands.xUnlockDoors := FALSE;

END_ACTION
```

#### ConsentLine.st - Consent Line
```iecst
ACTION ConsentsLine:
		(*
		View OF the machine from the Operator side

		>>>>>> LeftHandMachine 					RightHandMachine <<<<<<<<
		(BK_A #1 >> BK_B #2)		LOGICAL			(BK_A #2 << BK_B #1)

			          ################-################
		L2	          ################-################     L2
		------        ################-################   -------
		L1	          ################-################     L1
			##########################-###########################
			##########################-###########################
			    ######################-#######################
			    ######################-#######################
			    ######################-#######################
			    ######################-#######################

			BLOCK A [1-physical]				BLOCK B [2-physical]

		*)

	///////////////////////////////////////////////////
	// Consents depending if double or simple line
	//////////////////////////////////////////////////

	gDryer.In.xConsentOk := gDryer.St.Mode.xAuto;

	tonDelayConsentInput.IN:= gDryer.In.xConsentOk;
	tonDelayConsentInput.PT:= T#100ms;
	tonDelayConsentInput();

	gDryer.St.xConsent:= tonDelayConsentInput.Q;

	///////////////////////////////////////////////////////////////////////////////////////
	///////////////////////////////////////////////////////////////////////////////////////
	///////////////////////////////////////////////////////////////////////////////////////

	// Pending to test
	//Consent Outputs for L1
	//Single line L1, When belt is runing is because we had consent
	xOutputConsentInSingleLineL1:=	gDryer.In.xConsentOk AND gDryer.St.AutoMode.xProdORByPass AND NOT gThicknessCtrl.status.MediaPosition.xMountedMediaInside;

	xOutputConsentInByPassL1 := gDryer.St.AutoMode.xBypass AND gDryer.In.xConsentOk;

	//Consider the delay of the output signal configured in SW
	tonDelayConsentOutL1.IN:= gBelt.states.xRuningBelt AND (xOutputConsentInSingleLineL1 OR xOutputConsentInByPassL1);// It checked in both single or dtpL1
	tonDelayConsentOutL1.PT:= gDryer.Pt.SW.tiDelayConsent;
	tonDelayConsentOutL1();

	gDryer.Out.xConsentL1:= tonDelayConsentOutL1.Q;

END_ACTION
```

#### SuctionBlower.st
```iecst
ACTION SuctionBlower:

	////////////////////////////
	// BLOWERS
	////////////////////////////
	// Reference Jira: CRETAPRINT LEGOCRETALEGO-845
	// Turbine: Suction mode in automatic it isn´t correct.
	//
	// gui_i_iModoTurbina
	// Suction mode functionality. It can be configured by GUI with Ventrui or Turbine parameters
	// 0 estado off, 1 estado siempre On, modo 2, con base de tiempo en la desconexion.

	CASE gDryer.Pt.SW.Suction.iBlowerMode OF

		BWMODE_OFF:
			gDryer.Out.xSuctionTurbine:= FALSE;

		BWMODE_ON:
			gDryer.Out.xSuctionTurbine:= TRUE;

		BWMODE_AUTO:
			tofDelaySuction.IN:=gDryer.St.Mode.xAuto AND gBelt.states.xRuningBelt;
			tofDelaySuction.PT:=gDryer.Pt.SW.Suction.tiBlowerDelayOff;
			tofDelaySuction();

			gDryer.Out.xSuctionTurbine:= tofDelaySuction.Q;

	END_CASE;

END_ACTION
```

#### ResetRouterAndHub.st - Reset Router and CB 
```iecst
ACTION ResetRouterAndHub:

	// Reset Router
	tof_ResetSwitch.IN:=gDryer.commands.xResetSwitch;
	tof_ResetSwitch.PT:= T#6s;
	tof_ResetSwitch();
	gDryer.commands.xResetSwitch:= FALSE;

	gDryer.Out.xResetSwitch := tof_ResetSwitch.Q;

	// Reset Hub
	tof_ResetHub.IN:=gDryer.commands.xResetHub;
	tof_ResetHub.PT:= T#4s;
	tof_ResetHub();
	gDryer.commands.xResetHub:= FALSE;

	gDryer.Out.xResetHub := tof_ResetHub.Q;

	// Reset Fan Breaker
	tof_ResetFanBreaker.IN:=gDryer.commands.xResetFanBreaker;
	tof_ResetFanBreaker.PT:= T#2s;
	tof_ResetFanBreaker();
	gDryer.commands.xResetFanBreaker:= FALSE;

	gDryer.Out.xResetFanBreaker := tof_ResetFanBreaker.Q;

END_ACTION
```

#### OrdersSlow.st
```iecst
ACTION OrdersSlow:

	gThicknessCtrl.parameters.ContinuousMedia.MediaData.iLine := 1;
	gThicknessCtrl.parameters.ContinuousMedia.MediaData.rWidth := gDryer.Pt.SW.Media.rWidth;
	gThicknessCtrl.parameters.ContinuousMedia.MediaData.rLength := gDryer.Pt.SW.Media.rLength;
	gThicknessCtrl.parameters.ContinuousMedia.MediaData.rCrossOffset := gDryer.Pt.SW.Media.rCrossOffset;
	gThicknessCtrl.parameters.ContinuousMedia.MediaData.rDocWidth := gDryer.Pt.SW.Media.rDocWidth;
	gThicknessCtrl.parameters.ContinuousMedia.MediaData.rDocLength := gDryer.Pt.SW.Media.rDocLength;
	gThicknessCtrl.parameters.ContinuousMedia.MediaData.rDocCrossOffset := gDryer.Pt.SW.Media.rDocCrossOffset;

	IF gDryer.St.AutoLocation.xRemote THEN
		gThicknessCtrl.parameters.CheckMedia[1].xActive := gDryerRemoteData.Parameters.xPrinterBeltRuning AND NOT gDryerRemoteData.Parameters.xLineEmptyingBelt; //NOZOMITWO-2447
		gThicknessCtrl.parameters.CheckMedia[2].xActive := gDryerRemoteData.Parameters.xPrinterBeltRuning AND NOT gDryerRemoteData.Parameters.xLineEmptyingBelt AND gDryer.Pt.SW.xDoubleLine; //NOZOMITWO-2447
	ELSE
		gThicknessCtrl.parameters.CheckMedia[1].xActive := TRUE;								//NOZOMITWO-2424
		gThicknessCtrl.parameters.CheckMedia[2].xActive := gDryer.Pt.SW.xDoubleLine;			//NOZOMITWO-2424
	END_IF

	IF NOT gDryer.St.AutoLocation.xRemote THEN
		gDryer.Pt.SW.Media.rCrossOffset := (-1) * gDryer.Pt.SW.Media.rWidth / 2;
		gDryer.Pt.SW.Media.rDocLength := gDryer.Pt.SW.Media.rLength;
		gDryer.Pt.SW.Media.rDocWidth := gDryer.Pt.SW.Media.rWidth;
		gDryer.Pt.SW.Media.rDocCrossOffset := gDryer.Pt.SW.Media.rCrossOffset;
	END_IF

	ThermalInertia;

	IF gThicknessCtrl.parameters.Dry.iMinDryValue <= 0 THEN
		gThicknessCtrl.parameters.Dry.iMinDryValue := 8;
	END_IF

END_ACTION

ACTION ThermalInertia:

	/////////////////////////////////////////////////////////////////
	///// THERMAL INERTIA	THERMAL INERTIA		THERMAL INERTIA	/////
	/////////////////////////////////////////////////////////////////

	// Check initial data
	IF gDryer.Pt.ThermalInertia.iBoardsToStartReducing = 0 OR
		gDryer.Pt.ThermalInertia.iBoardsToMaxPowerReduction = 0 OR
		gDryer.Pt.ThermalInertia.iBoardsToStartReducing >= gDryer.Pt.ThermalInertia.iBoardsToMaxPowerReduction OR
		gDryer.Pt.ThermalInertia.rMaxPowerReduction > 1 THEN

				rThermalInerciaReduction := 1;
				gThicknessCtrl.parameters.Dry.rThermalInerciaReduction := rThermalInerciaReduction;
				RETURN;
	END_IF

	// Initial data and step calculation
	IF NOT gNirAdphos.Signals.Out.xProcess THEN
		rThermalInerciaReduction := 1;
		rThermalInerciaStepReduction := (1- gDryer.Pt.ThermalInertia.rMaxPowerReduction)/(gDryer.Pt.ThermalInertia.iBoardsToMaxPowerReduction - gDryer.Pt.ThermalInertia.iBoardsToStartReducing);
		iBoardsAtStartDryingL1 := gThicknessCtrl.status.Detection.iBoardsFromStartL1;
	END_IF

	iBoardsFromStartL1 := gThicknessCtrl.status.Detection.iBoardsFromStartL1 - iBoardsAtStartDryingL1;

	IF iBoardsFromStartL1 > gDryer.Pt.ThermalInertia.iBoardsToStartReducing AND iBoardsFromStartL1 <= gDryer.Pt.ThermalInertia.iBoardsToMaxPowerReduction THEN
		rThermalInerciaReduction := 1 - rThermalInerciaStepReduction * (iBoardsFromStartL1 - gDryer.Pt.ThermalInertia.iBoardsToStartReducing);
	ELSIF iBoardsFromStartL1 > gDryer.Pt.ThermalInertia.iBoardsToMaxPowerReduction THEN
		rThermalInerciaReduction := gDryer.Pt.ThermalInertia.rMaxPowerReduction;
	END_IF

	gThicknessCtrl.parameters.Dry.rThermalInerciaReduction := rThermalInerciaReduction;

END_ACTION
```

#### LightBeacon.st - External light beacon
```iecst
ACTION LightBeacon:

	// Red: Safety related alarm
	iReasonRedLight.0 := gDryer.AlSummary.xAlrSafetySystemGeneral;
	gDryer.Out.xRedLight := iReasonRedLight>0;

	// Yellow Blinking: stop or critical alarm
	iReasonBlinkYellowLight.0 := gDryer.AlSummary.xAlarmCritical;
	iReasonBlinkYellowLight.1 := gDryer.AlSummary.xAlarmStop;
	// Yellow Solid: warning
	iReasonSolidYellowLight.0 := gDryer.AlSummary.xAnyWarning;

	IF (iReasonBlinkYellowLight > 0) THEN
		gDryer.Out.xYellowLight := gPLC.xBlk_1s;
	ELSIF (iReasonSolidYellowLight > 0) THEN
		gDryer.Out.xYellowLight := TRUE;
	ELSE
		gDryer.Out.xYellowLight := FALSE;
	END_IF

	// Blue: Any alarm may be reset
	iReasonBlueLight.0 := (NOT gDryer.AlSummary.xAlarmCritical) AND (gDryer.AlSummary.iReasonCritical > 0);
	iReasonBlueLight.1 := (NOT gDryer.AlSummary.xAlarmStop) AND (gDryer.AlSummary.iReasonStop[0] > 0);
	iReasonBlueLight.2 := (NOT gDryer.Al.xAlrStopDrying) AND (gDryer.Al.iReasonStopDrying > 0);
	gDryer.Out.xBlueLight := iReasonBlueLight > 0;

	// White: Automatic and remote mode
	iReasonWhiteLight.0 := gDryer.St.AutoLocation.xRemote; //NOZDRYER-381
	gDryer.Out.xWhiteLight := iReasonWhiteLight > 0;

	////////////////////////////
	// LIGHT RESET
	////////////////////////////
	gDryer.Out.xLightReset:= gDryer.AutoCmd.xReset;

END_ACTION
```

#### DryerCtrl_Slow.var - Local variables
```iecst
VAR
	arAnyStopAlarmMuted : AutoResetSound;
	arFanBreakers : AutoResetSound;
	arFan24Vdc : AutoResetSound;
	arMain24Vdc : AutoResetSound;
	arBentTile : AutoResetSound;
	arWrongPhysConf : AutoResetSound;
	arAnyJam : AutoResetSound;
	arBentMedia : AutoResetSound;
	arPDSensorErrorL1 : AutoResetSound;
	arPDSensorErrorL2 : AutoResetSound;
	Blink_1s : Blink;
	Blink_2s : Blink;
	Blink_5s : Blink;
	Blink_100ms : Blink;
	Blink_200ms : Blink;
	Blink_500ms : Blink;
	xAllBlocksCleaning : BOOL;
	xInstantPrintL2 : BOOL;
	xAllBlocksCleaningEnded : BOOL;
	xInstantPrintL1 : BOOL; (*command bool edge*)
	xCleanOrderBK2 : BOOL := FALSE;
	xShotLine2 : BOOL;
	xRobotReadyToPrint : BOOL;
	xCleanOrderBK1 : BOOL := FALSE;
	xCleanSequencially : BOOL := FALSE;
	testCanOpen : BOOL;
	xShotLine1 : BOOL;
	xOrderToGap : BOOL;
	xCleanBeltForced : BOOL;
	xCleaningBeltByTiles : BOOL;
	xOutputConsentInSingleLineL1 : BOOL;
	xOutputConsentInByPassL1 : BOOL;
	xOutputConsentInByPassL2 : BOOL;
	xOnPcs : BOOL;
	xCleaningBeltByTime : BOOL;
	xCleanBeltOrder : BOOL; (*Internal to assign cleaning belt system *)
	FbCleanDelayControl_1 : FbCleanDelayControl;
	RTInfo_0 : RTInfo;
	tof_ResetHub : TOF;
	tof_ResetFanBreaker : TOF;
	tofCleaningTrayBelt : TOF;
	tofDelaySuction : TOF; (*tiMinutes : TIME;*)
	tof_ResetSwitch : TOF;
	T_OnPcs : TON;
	tonCleaningByTime : TON;
	T_BtwnCleans : TON;
	tonDelayConsentInput : TON;
	tonCleanbyTime : TON;
	tonDelayConsentOutL2 : TON;
	tonDelayConsentOutL1 : TON;
	tonCleaningBelt : TON;
	tonCleanBelt : TON;
	iIndexInks : USINT; (*Inks Index to use a FOR*)
	iIndexBlock : USINT; (*Block Index to use a FOR*)
	tiCleaningBeltByTime : TIME;
	iSPTilesToCleanBelt : INT;
	xAnyBlockToPrint : BOOL;
	reasonSoundGen : UDINT;
	reasonBuzzer : UDINT;
	iIndex : USINT; (*FOR index*)
	iBentMediaCounter : UINT; (*Counter of bent media. Just for the alarm of max movements*)
	tonDecreaseMovCount : TON; (*Time to decrease the count of max movements*)
	tonStartSound : TON;
	iCountStartSound : USINT;
	xStartSound : BOOL;
	strAux : STRING[80];
	plcCardsOK : UDINT;
	iReasonLockDoors : UINT;
	iReasonReleaseDoors : UINT;
	iReasonRedLight : UINT;
	iReasonBlinkYellowLight : UINT;
	iReasonSolidYellowLight : UINT;
	iReasonBlueLight : UINT;
	iReasonWhiteLight : UINT;
	xReleaseDoors : BOOL;
	xLockDoors : BOOL;
	tonBeltOvertorque : TON;
	tonBeltOverTempFast : TON;
	tonBeltOverTempSlow : TON;
	rThermalInerciaReduction : REAL;
	rThermalInerciaStepReduction : REAL;
	iBoardsAtStartDryingL1 : UDINT;
	iBoardsFromStartL1 : UDINT;
END_VAR
```

- CleaningStates.graphml - YED documentation (not shown)

### Package Logical/Dryer/PhysicalMapping - Physical inputs assignation

### Program Logical/Dryer/PhysicalMapping/PhysicalMapInputs (IEC) - Inputs program

#### InputsDryerNoz2.st - PhysicalInputs
```iecst
ACTION InputsDryerNoz2:

	//REMOTE SIGNALS
	gDryer.In.Safety := gDryerRemoteData.Signals.Safety;
	tonNoCommsPrinter.IN := NOT gDryerRemoteData.xCommsOK;
	tonNoCommsPrinter.PT := t#1s;
	tonNoCommsPrinter();
	IF gDryerRemoteData.xCommsOK THEN
		gAxisInverter[1].ElecSignals.In.xBreakerOK := gDryerRemoteData.Signals.xBreakerOKBlowerInput; //NOT Line_X20DIF371_003.DInput[15];
	ELSIF tonNoCommsPrinter.Q THEN
		gAxisInverter[1].ElecSignals.In.xBreakerOK := FALSE;
	END_IF

	gAxisInverter[2].ElecSignals.In.xBreakerOK := gDryerRemoteData.Signals.xBreakerOKBlowerOutput; //NOT Line_X20DIF371_003.DInput[16];

	// X20DIF371_201 DIGITAL INPUTS
	gBasicDetectMedia.Inputs.xMountedMedia := NOT X20DIF371_201.DInput[1];
	gDryer.In.Buttons.xStop := NOT X20DIF371_201.DInput[2];
	gDryer.In.Buttons.xReset := X20DIF371_201.DInput[3];
	gDryer.In.xFanBreakersOK := X20DIF371_201.DInput[4];
	gDryer.In.xFanBreakersWarning := X20DIF371_201.DInput[5];
	gDryer.In.xOpenDoorsKey := X20DIF371_201.DInput[6];
	gSimpleBlock[1].In.xReferenceDI := X20DIF371_201.DInput[7];
	//gBasicDetectMedia.Inputs.xCorrection := NOT X20DIF371_201.DInput[8];
	gDryer.In.xFan24VdcOK := X20DIF371_201.DInput[9];
	gDryer.In.xMain24VdcOK := X20DIF371_201.DInput[10];

	gDryer.In.iMachineModelCode.0 := X20DIF371_201.DInput[13];
	gDryer.In.iMachineModelCode.1 := X20DIF371_201.DInput[14];
	gDryer.In.iMachineModelCode.2 := X20DIF371_201.DInput[15];
	gDryer.In.iMachineModelCode.3 := X20DIF371_201.DInput[16];

	// X20DIF371_202 DIGITAL INPUTS
	gNirAdphos.Signals.In.xReady:= X20DIF371_202.DInput[1];
	gNirAdphos.Signals.In.xInProcess := X20DIF371_202.DInput[2];
	gNirAdphos.Signals.In.xFault := X20DIF371_202.DInput[3];
	gDryerRemoteData.Commands.xRunTransport := X20DIF371_202.DInput[4];
	gDryer.In.Buttons.xAuto := gDryer.In.xAuto_GI := X20DIF371_202.DInput[5];
	gDryer.In.Buttons.xZero := gDryer.In.xZero_GI := NOT X20DIF371_202.DInput[6];
	gDryer.In.Buttons.xManual := gDryer.In.xManual_GI := X20DIF371_202.DInput[7];
	gDryer.In.Buttons.xStopBlowers := X20DIF371_202.DInput[8];
	gNirAdphos.Signals.In.Jam[2].xMechCross := NOT X20DIF371_202.DInput[9] OR NOT X20DIF371_202.DInput[10];
	gBasicDetectMedia.Inputs.xMediaPresentL1 := X20DIF371_202.DInput[13] AND (NOT gDryer.St.AutoLocation.xRemote OR gDryerRemoteData.Parameters.xPrinterBeltRuning); //NOZOMITWO-2512
	gThicknessCtrl.Inputs.CheckMedia[1].xCheckFail := X20DIF371_202.DInput[14];
	gBasicDetectMedia.Inputs.xMediaPresentL2 := X20DIF371_202.DInput[15];
	gThicknessCtrl.Inputs.CheckMedia[2].xCheckFail := X20DIF371_202.DInput[16];

	// X20DIF371_203 DIGITAL INPUTS
	gNirAdphos.Signals.In.BlockedFans[1].Fan[1]	:= X20DIF371_203.DInput[1];
	gNirAdphos.Signals.In.BlockedFans[1].Fan[2]	:= X20DIF371_203.DInput[2];
	gNirAdphos.Signals.In.BlockedFans[1].Fan[3]	:= X20DIF371_203.DInput[3];
	gNirAdphos.Signals.In.BlockedFans[1].Fan[4]	:= X20DIF371_203.DInput[4];

	gNirAdphos.Signals.In.BlockedFans[2].Fan[1]	:= X20DIF371_203.DInput[5];
	gNirAdphos.Signals.In.BlockedFans[2].Fan[2]	:= X20DIF371_203.DInput[6];
	gNirAdphos.Signals.In.BlockedFans[2].Fan[3]	:= X20DIF371_203.DInput[7];
	gNirAdphos.Signals.In.BlockedFans[2].Fan[4]	:= X20DIF371_203.DInput[8];

	gJamDetect[1].Inputs.xJamCrash[1] := X20DIF371_203.DInput[9];
	gJamDetect[1].Inputs.xJamCrash[2] := X20DIF371_203.DInput[10];
	gJamDetect[1].Inputs.xJamCrash[3] := X20DIF371_203.DInput[11];
	gJamDetect[1].Inputs.xJamCrash[4] := X20DIF371_203.DInput[12];
	gJamDetect[1].Inputs.xJamLowCrash := X20DIF371_203.DInput[13];
	gJamDetect[1].Inputs.xJamTestOk := X20DIF371_203.DInput[14];

	gNirAdphos.Signals.In.Jam[1].xMechCross := NOT X20DIF371_203.DInput[15] OR NOT X20DIF371_203.DInput[16];

	// X20AI8321_207 ANALOG INPUTS
	gDryer.In.Temp.iBoardInRaw := X20AI8321_207.AInput[1];
	gDryer.In.Temp.iBoardOutRaw := X20AI8321_207.AInput[2];
	gDryer.In.Temp.iBeltRaw := X20AI8321_207.AInput[3];
	gNirAdphos.Signals.In.iInletHumidityRaw := X20AI8321_207.AInput[4];
	gNirAdphos.Signals.In.iInletTempRaw := X20AI8321_207.AInput[5];
	gTransVacuum[1].Inputs.iPressureRaw := X20AI8321_207.AInput[6];
	gDryer.In.Temp.iAirBlowerInputRaw := X20AI8321_207.AInput[7];
	gDryer.In.Temp.iAirBlowerOutputRaw := X20AI8321_207.AInput[8];

	gDryer.In.Temp.xBoardInSensorError := StatusAnalogInputBroken( X20AI8321_207.ModuleOk, X20AI8321_207.Status01, X20AI8321_207.Status02, 1);
	gDryer.In.Temp.xBoardOutSensorError := StatusAnalogInputBroken( X20AI8321_207.ModuleOk, X20AI8321_207.Status01, X20AI8321_207.Status02, 2);
	gDryer.In.Temp.xBeltSensorError := StatusAnalogInputBroken( X20AI8321_207.ModuleOk, X20AI8321_207.Status01, X20AI8321_207.Status02, 3);
	gNirAdphos.Signals.In.xInletHumiditySensorError := StatusAnalogInputBroken( X20AI8321_207.ModuleOk, X20AI8321_207.Status01, X20AI8321_207.Status02, 4);
	gNirAdphos.Signals.In.xInletTempSensorError := StatusAnalogInputBroken( X20AI8321_207.ModuleOk, X20AI8321_207.Status01, X20AI8321_207.Status02, 5);
	gTransVacuum[1].Inputs.xPressureSensorError	:= StatusAnalogInputBroken(X20AI8321_207.ModuleOk, X20AI8321_207.Status01, X20AI8321_207.Status02, 6);
	gDryer.In.Temp.xAirBlowerInputSensorError := StatusAnalogInputBroken( X20AI8321_207.ModuleOk, X20AI8321_207.Status01, X20AI8321_207.Status02, 7);
	gDryer.In.Temp.xAirBlowerOutputSensorError := StatusAnalogInputBroken( X20AI8321_207.ModuleOk, X20AI8321_207.Status01, X20AI8321_207.Status02, 8);

	// X20AT4222_209 TEMPERATURE INPUTS
	gNirAdphos.Signals.In.iSurfaceTempModuleRaw[1] := X20AT4222_209.TempInput[1];
	gNirAdphos.Signals.In.iSurfaceTempModuleRaw[2] := X20AT4222_209.TempInput[2];

	gNirAdphos.Signals.In.xSurfaceTempModuleSensorError[1] := StatusAnalogInputBroken( X20AT4222_209.ModuleOk, X20AT4222_209.Status01, X20AT4222_209.Status02, 1);
	gNirAdphos.Signals.In.xSurfaceTempModuleSensorError[2] := StatusAnalogInputBroken( X20AT4222_209.ModuleOk, X20AT4222_209.Status01, X20AT4222_209.Status02, 2);

END_ACTION
```

#### Variables.var - Local variables
```iecst
VAR
	T_Mute : TOF;
	T_Reset : TON;
	iIndexBlock : USINT;
	tonNoCommsPrinter : TON;
END_VAR
```

### Program Logical/Dryer/PhysicalMapping/PhysicalMapOutputs (IEC) - Physical outputs assignation

#### MappingOutputs.st - PhysicalInputs
```iecst
PROGRAM _CYCLIC

	CASE gDryer.Pt.MachineModel OF
		DryerType_NOZ2_NIR,
		DryerType_NOZ2_NIR_ARCLAMP:
			OutputsDryerNoz2;

	END_CASE

END_PROGRAM
```

### SimDryer.var
```iecst
VAR
	iSimIndex : USINT; (*Index for loops in simulation*)
	simEventLog : EventLog_typ;
	webClient : httpClient;
	ResponseHeader : httpResponseHeader_t;
	RequestData : STRING[3000];
	ResponseData : STRING[3000];
	URLHost : STRING[80];
	URIHost : STRING[80];
	xTestPrepareDryer : BOOL; (*This value must be used as active while pressed by the visualization*)
	xTestBeltTests : BOOL; (*This value must be used as active while pressed by the visualization*)
	xTestConsents : BOOL; (*This value must be used as active while pressed by the visualization*)
	xTestLine : BOOL; (*This value must be used as active while pressed by the visualization*)
	xTestCleaning : BOOL; (*This value must be used as active while pressed by the visualization*)
	testMonitor : UtMgrMonitor;
	simMachineType : INT;
	simMachineTypeCopy : INT;
	simMachineTypeEnumCopy : SimMachineType;
	xSimulateMedia : BOOL;
	tonSimMedia : TON;
	tonSimMediaAuto : TON;
END_VAR
```

- DryerConection.uap (not shown)

- Program Logical/Dryer/DryerSimAnc/DryerSimAnc_v1/DryerSimAnc (IEC) (no source held here)

### DryerSimAnc.typ
```iecst
TYPE
	DryerSimCommands_typ : 	STRUCT
		CreateError : BOOL;
	END_STRUCT;
	DryerSimAnc_typ : 	STRUCT
		Commands : DryerSimCommands_typ;
	END_STRUCT;
END_TYPE
```

### Package Logical/AxisTables - Axis table configuration

### Data object Logical/AxisTables/AcpErrTxt (Ett)

- AcpErrTxt.ett (not shown)

### Data object Logical/AxisTables/acp10etxen (Ett)

- acp10etxen.ett (not shown)

### Data object Logical/AxisTables/SM_a (Apt) - Stepper Motors 3 Lasers config table

#### SM_a.apt
```
AcoposParameterTable:
  Root Parameters:
    64232 = 25600 (Name=SM_SCALE_STEP)
    64233 = 1000 (Name=SM_SCALE_LOAD_UNITS)
    64234 = 1 (Name=SM_SCALE_LOAD_MOTREV)
    109 = 1024 (Name=SCALE_ENCOD_INCR)
    128 = 1 (Name=SGEN_SW_END_IGNORE)  // Limit values: Ignore SW end positions
```

- Data object Logical/AxisTables/SM_i (Ax) - Stepper Motors 3 Lasers config table (no source held here)

### Data object Logical/AxisTables/BeltP4_a (Apt)

#### BeltA.apt
```
AcoposParameterTable:
  Root Parameters:
    128 = 1 (Name=SGEN_SW_END_IGNORE)  // Limit values: Ignore SW end positions
```

- Data object Logical/AxisTables/BeltP4_i (Ax) (no source held here)

- Data object Logical/AxisTables/BeltCube_a (Apt) (no source held here)

### Data object Logical/AxisTables/BeltCube_i (Ax)

#### BeltI.ax
```
InitParameter (Version=5.21.2, NcSwId=ACP10)
  ACP10AXIS_typ:
    dig_in:
      level:
        reference = ncACTIV_LO
        pos_hw_end = ncACTIV_HI
        neg_hw_end = ncACTIV_HI
        trigger1 = ncACTIV_LO
        trigger2 = ncACTIV_LO
    encoder_if:
      parameter:
        count_dir = ncSTANDARD
        scaling:
          load:
            units = 1000
            rev_motor = 1
    limit:
      parameter:
        v_pos = 435800.0
        v_neg = 435800.0
        a1_pos = 1400000.0
        a2_pos = 1400000.0
        a1_neg = 1400000.0
        a2_neg = 1400000.0
        t_jolt = 0.0
        t_in_pos = 0.0
        pos_sw_end = 8388607
        neg_sw_end = -8388608
        ds_warning = 500.0
        ds_stop = 1000.0
        a_stop = 6.53E+07
        dv_stop = 0.0
        dv_stop_mode = ncOFF
    controller:
      mode = ncPOSITION
      position:
        kv = 376.0
        tn = 0.0
        t_predict = 0.0004
        t_total = 0.0004
        p_max = 1.0E+30
        i_max = 0.0
      speed:
        kv = 25.3
        tn = 0.0
        t_filter = 0.0
        isq_filter1:
          type = ncOFF
          a0 = 0.0
          a1 = 0.0
          b0 = 0.0
          b1 = 0.0
          b2 = 0.0
          c0_par_id = 0
          c1_par_id = 0
        isq_filter2:
          type = ncOFF
          a0 = 0.0
          a1 = 0.0
          b0 = 0.0
          b1 = 0.0
          b2 = 0.0
          c0_par_id = 0
          c1_par_id = 0
        isq_filter3:
          type = ncOFF
          a0 = 0.0
          a1 = 0.0
          b0 = 0.0
          b1 = 0.0
          b2 = 0.0
          c0_par_id = 0
          c1_par_id = 0
      uf:
        type = ncLINEAR
        auto_config = ncMOTOR_PAR
        u0 = 0.0
        un = 0.0
        fn = 50.0
        k_f_slip = 0.0
      ff:
        mode = ncSTANDARD
        torque_load = 0.0
        torque_pos = 0.0
        torque_neg = 0.0
        kv_torque = 0.0
        inertia = 0.0
        t_filter_a = 0.0
      fb:
        mode = ncSTANDARD
        speed_mix_ratio = 0.0
        speed_kv = 0.0
      model:
        mass1:
          inertia = 0.0
          viscous_friction = 0.0
        mass2:
          inertia = 0.0
          viscous_friction = 0.0
          stiffness = 0.0
          damping = 0.0
    move:
      stop:
        parameter[0]:
          decel_ramp = ncA_LIMIT
          controller = ncON
        parameter[1]:
          decel_ramp = ncA_LIMIT
          controller = ncON
        parameter[2]:
          decel_ramp = ncA_LIMIT
          controller = ncON
        parameter[3]:
          decel_ramp = ncA_LIMIT
          controller = ncON
        quickstop:
          decel_ramp = ncA_LIMIT
          t_jolt = 0.0
        drive_error:
          decel_ramp = ncA_LIMIT
      homing:
        parameter:
          s = 0
          v_switch = 5000.0
          v_trigger = 500.0
          a = 50000.0
          mode = ncDIRECT
          edge_sw = ncPOSITIVE
          start_dir = ncPOSITIVE
          trigg_dir = ncPOSITIVE
          ref_pulse = ncOFF
          fix_dir = ncOFF
          tr_s_block = 0.0
          torque_lim = 0.0
          ds_block = 0.0
          ds_stop = 0.0
      basis:
        parameter:
          v_pos = 5000.0
          v_neg = 5000.0
          a1_pos = 50000.0
          a2_pos = 50000.0
          a1_neg = 50000.0
          a2_neg = 50000.0
    message:
      text:
        parameter:
          format = ncBREAK
          columns = 80
          data_modul = acp10etxen
```

### Data object Logical/AxisTables/BeltP5_i (Ax)

#### BeltI.ax
```
InitParameter (Version=5.11.1, NcSwId=ACP10)
  ACP10AXIS_typ:
    dig_in:
      level:
        reference = ncACTIV_LO
        pos_hw_end = ncACTIV_HI
        neg_hw_end = ncACTIV_HI
        trigger1 = ncACTIV_LO
        trigger2 = ncACTIV_LO
    encoder_if:
      parameter:
        count_dir = ncSTANDARD
        scaling:
          load:
            units = 1000
            rev_motor = 1
    limit:
      parameter:
        v_pos = 435800.0
        v_neg = 435800.0
        a1_pos = 653000.0
        a2_pos = 653000.0
        a1_neg = 653000.0
        a2_neg = 653000.0
        t_jolt = 0.0
        t_in_pos = 0.0
        pos_sw_end = 8388607
        neg_sw_end = -8388608
        ds_warning = 500.0
        ds_stop = 1000.0
        a_stop = 6.53E+07
        dv_stop = 0.0
        dv_stop_mode = ncOFF
    controller:
      mode = ncPOSITION
      position:
        kv = 446.0
        tn = 0.0
        t_predict = 0.0004
        t_total = 0.0004
        p_max = 1.0E+30
        i_max = 0.0
      speed:
        kv = 11.7
        tn = 0.0
        t_filter = 0.0
        isq_filter1:
          type = ncOFF
          a0 = 0.0
          a1 = 0.0
          b0 = 0.0
          b1 = 0.0
          b2 = 0.0
          c0_par_id = 0
          c1_par_id = 0
        isq_filter2:
          type = ncOFF
          a0 = 0.0
          a1 = 0.0
          b0 = 0.0
          b1 = 0.0
          b2 = 0.0
          c0_par_id = 0
          c1_par_id = 0
        isq_filter3:
          type = ncOFF
          a0 = 0.0
          a1 = 0.0
          b0 = 0.0
          b1 = 0.0
          b2 = 0.0
          c0_par_id = 0
          c1_par_id = 0
      uf:
        type = ncLINEAR
        auto_config = ncMOTOR_PAR
        u0 = 0.0
        un = 0.0
        fn = 50.0
        k_f_slip = 0.0
      ff:
        mode = ncSTANDARD
        torque_load = 0.0
        torque_pos = 0.0
        torque_neg = 0.0
        kv_torque = 0.0
        inertia = 0.0
        t_filter_a = 0.0
      fb:
        mode = ncSTANDARD
        speed_mix_ratio = 0.0
        speed_kv = 2.0
      model:
        mass1:
          inertia = 0.0
          viscous_friction = 0.0
        mass2:
          inertia = 0.0
          viscous_friction = 0.0
          stiffness = 0.0
          damping = 0.0
    move:
      stop:
        parameter[0]:
          decel_ramp = ncA_LIMIT
          controller = ncON
        parameter[1]:
          decel_ramp = ncA_LIMIT
          controller = ncON
        parameter[2]:
          decel_ramp = ncA_LIMIT
          controller = ncON
        parameter[3]:
          decel_ramp = ncA_LIMIT
          controller = ncON
        quickstop:
          decel_ramp = ncA_LIMIT
          t_jolt = 0.0
        drive_error:
          decel_ramp = ncA_LIMIT
      homing:
        parameter:
          s = 0
          v_switch = 5000.0
          v_trigger = 500.0
          a = 50000.0
          mode = ncDIRECT
          edge_sw = ncPOSITIVE
          start_dir = ncPOSITIVE
          trigg_dir = ncPOSITIVE
          ref_pulse = ncOFF
          fix_dir = ncOFF
          tr_s_block = 0.0
          torque_lim = 0.0
          ds_block = 0.0
          ds_stop = 0.0
      basis:
        parameter:
          v_pos = 5000.0
          v_neg = 5000.0
          a1_pos = 50000.0
          a2_pos = 50000.0
          a1_neg = 50000.0
          a2_neg = 50000.0
    message:
      text:
        parameter:
          format = ncBREAK
          columns = 80
          data_modul = acp10etxen
```

### Data object Logical/AxisTables/BK1_a (Apt)

#### BK1_a.apt
```
AcoposParameterTable:
  Root Parameters
```

- Data object Logical/AxisTables/BK_sim_a (Apt) (no source held here)

- Data object Logical/AxisTables/NonCrash_a (Apt) (no source held here)

- Data object Logical/AxisTables/BK1_S1400_a (Apt) (no source held here)

### Data object Logical/AxisTables/BK1_S1400_i (Ax)

#### BK1_i.ax
```
InitParameter (Version=5.18.1, NcSwId=ACP10)
  ACP10AXIS_typ:
    dig_in:
      level:
        reference = ncACTIV_LO
        pos_hw_end = ncACTIV_HI
        neg_hw_end = ncACTIV_HI
        trigger1 = ncACTIV_HI
        trigger2 = ncACTIV_HI
    encoder_if:
      parameter:
        count_dir = ncSTANDARD
        scaling:
          load:
            units = 1000
            rev_motor = 1
    limit:
      parameter:
        v_pos = 100000.0
        v_neg = 100000.0
        a1_pos = 725000.0
        a2_pos = 725000.0
        a1_neg = 725000.0
        a2_neg = 725000.0
        t_jolt = 0.0
        t_in_pos = 0.0
        pos_sw_end = 700000
        neg_sw_end = -700000
        ds_warning = 500.0
        ds_stop = 1000.0
        a_stop = 725000.0
        dv_stop = 0.0
        dv_stop_mode = ncOFF
    controller:
      mode = ncPOSITION
      position:
        kv = 160.0
        tn = 0.0
        t_predict = 0.0004
        t_total = 0.0004
        p_max = 1.0E+30
        i_max = 0.0
      speed:
        kv = 1.15
        tn = 0.0
        t_filter = 0.0
        isq_filter1:
          type = ncOFF
          a0 = 0.0
          a1 = 0.0
          b0 = 0.0
          b1 = 0.0
          b2 = 0.0
          c0_par_id = 0
          c1_par_id = 0
        isq_filter2:
          type = ncOFF
          a0 = 0.0
          a1 = 0.0
          b0 = 0.0
          b1 = 0.0
          b2 = 0.0
          c0_par_id = 0
          c1_par_id = 0
        isq_filter3:
          type = ncOFF
          a0 = 0.0
          a1 = 0.0
          b0 = 0.0
          b1 = 0.0
          b2 = 0.0
          c0_par_id = 0
          c1_par_id = 0
      uf:
        type = ncLINEAR
        auto_config = ncMOTOR_PAR
        u0 = 0.0
        un = 0.0
        fn = 50.0
        k_f_slip = 0.0
      ff:
        mode = ncSTANDARD
        torque_load = 0.0
        torque_pos = 0.0
        torque_neg = 0.0
        kv_torque = 0.0
        inertia = 0.0
        t_filter_a = 0.0
      fb:
        mode = ncSTANDARD
        speed_mix_ratio = 0.0
        speed_kv = 2.0
      model:
        mass1:
          inertia = 0
          viscous_friction = 0
        mass2:
          inertia = 0
          viscous_friction = 0
          stiffness = 0
          damping = 0
    move:
      stop:
        parameter[0]:
          decel_ramp = ncA_LIMIT
          controller = ncON
        parameter[1]:
          decel_ramp = ncA_LIMIT
          controller = ncON
        parameter[2]:
          decel_ramp = ncA_LIMIT
          controller = ncON
        parameter[3]:
          decel_ramp = ncA_LIMIT
          controller = ncON
        quickstop:
          decel_ramp = ncA_LIMIT
          t_jolt = 0.0
        drive_error:
          decel_ramp = ncA_LIMIT
      homing:
        parameter:
          s = 23200
          v_switch = 5000.0
          v_trigger = 500.0
          a = 50000.0
          mode = ncABS_SWITCH
          edge_sw = ncPOSITIVE
          start_dir = ncNEGATIVE
          trigg_dir = ncNEGATIVE
          ref_pulse = ncOFF
          fix_dir = ncOFF
          tr_s_block = 0.0
          torque_lim = 0.0
          ds_block = 0.0
          ds_stop = 0.0
      basis:
        parameter:
          v_pos = 5000.0
          v_neg = 5000.0
          a1_pos = 50000.0
          a2_pos = 50000.0
          a1_neg = 50000.0
          a2_neg = 50000.0
    message:
      text:
        parameter:
          format = ncBREAK
          columns = 80
          data_modul = acp10etxen
```

### Data object Logical/AxisTables/BK1_Cube_a (Apt)

#### BK1_a.apt
```
AcoposParameterTable:
  Root Parameters:
    944 = STAT_TRIGGER1 (Name=REFERENCE_SWITCH_PARID)  // Digital inputs: Parameter ID for reference switch
```

- Data object Logical/AxisTables/BK1_Cube_i (Ax) (no source held here)

### Data object Logical/AxisTables/BeltNozomi2_a (Apt)

#### BeltA.apt
```
AcoposParameterTable:
  Root Parameters:
    128 = 1 (Name=SGEN_SW_END_IGNORE)  // Limit values: Ignore SW end positions
    10 = 47 (Name=R_BLEEDER_EXT, Unit=Ohm)  // Bleeder: External: Resistance
    11 = 300 (Name=TEMP_MAX_BLEEDER_EXT, Unit=°C)  // Bleeder: External: Limit temperature
    12 = 0.93 (Name=RTH_BLEEDER_AMB_EXT, Unit=K/W)  // Bleeder: External: Thermal resistance
    13 = 30.82 (Name=CTH_BLEEDER_EXT, Unit=Ws/K)  // Bleeder: External: Thermal capacity
    398 = 1 (Name=BLEEDER_SELECTOR_EXT)  // Bleeder: Selector
```

### Data object Logical/AxisTables/Belt17000_a (Apt)

#### BeltA.apt
```
AcoposParameterTable:
  Root Parameters:
    128 = 1 (Name=SGEN_SW_END_IGNORE)  // Limit values: Ignore SW end positions
    10 = 47 (Name=R_BLEEDER_EXT, Unit=Ohm, Disabled=FALSE)  // Bleeder: External: Resistance
    11 = 300 (Name=TEMP_MAX_BLEEDER_EXT, Unit=°C, Disabled=FALSE)  // Bleeder: External: Limit temperature
    12 = 1.4 (Name=RTH_BLEEDER_AMB_EXT, Unit=K/W, Disabled=FALSE)  // Bleeder: External: Thermal resistance
    13 = 30.82 (Name=CTH_BLEEDER_EXT, Unit=Ws/K, Disabled=FALSE)  // Bleeder: External: Thermal capacity
    398 = 1 (Name=BLEEDER_SELECTOR_EXT, Disabled=FALSE)  // Bleeder: Selector
```

### Data object Logical/AxisTables/BK_17000_a (Apt)

#### BK_a.apt
```
AcoposParameterTable:
  Root Parameters:
    944 = STAT_TRIGGER1 (Name=REFERENCE_SWITCH_PARID)  // Digital inputs: Parameter ID for reference switch
```

### Package Logical/InkBox - Project Ink box external

- RunTextScript.bat (not shown)

### Program Logical/InkBox/Config/SavePermanent (IEC)

#### SavePermanent.var
```iecst
VAR
	iInksIndex : USINT;
END_VAR
```

- InksTextsAndAlarms.csv (not shown)

### Program Logical/InkBox/HMI/HMI (IEC)

#### HMI.st - Init, cyclic, exit code
```iecst
PROGRAM _INIT

	//This is to assure raise alarms started with TRUE
	MpViewAlarms;
	Alarms;

	iInkHMI_copy := 0;
END_PROGRAM

PROGRAM _CYCLIC

	// Pointer assignation and avoid out of range. 1 is the default one
	IF iInkHMI >= 1 AND iInkHMI <= MAX_LAST_INK THEN
		dataInksHMI ACCESS ADR(gInks[iInkHMI]);

		// Take the string value when changing system
		IF iInkHMI <> iInkHMI_copy THEN
			brsitoa(INT_TO_DINT(dataInksHMI.parSw.Config.iInkType), ADR(strInkType));
			brsitoa(INT_TO_DINT(dataInksHMI.parSw.Config.iPrintHeadType), ADR(strPrintHeadType));
		END_IF

		// Update value
		dataInksHMI.parSw.Config.iInkType := DINT_TO_INT(brsatoi(ADR(strInkType)));
		dataInksHMI.parSw.Config.iPrintHeadType := DINT_TO_INT(brsatoi(ADR(strPrintHeadType)));

		iInkHMI_copy := iInkHMI;
	ELSE
		iInkHMI := 1;
	END_IF

	MpViewAlarms;

	Alarms;

END_PROGRAM

PROGRAM _EXIT

	//Cards of the Ink Box
	X20DIF371_101;
	X20AI4322_102;
	X20AT2222_103;
	X20DOF322_104;
	X20AO4622_105;

	X20DIF371_201;
	X20AI4322_202;
	X20AT2222_203;
	X20DOF322_204;
	X20AO4622_205;

	X20DIF371_301;
	X20AI4322_302;
	X20AT2222_303;
	X20DOF322_304;
	X20AO4622_305;

END_PROGRAM
```

#### MpViewAlarms.st
```iecst
ACTION MpViewAlarms:

	AlarmsCore.Enable := TRUE;
	AlarmsCore.MpLink := ADR(gAlrCore);
	AlarmsCore();

	AlarmsHistory.Enable := TRUE;
	AlarmsHistory.MpLink := ADR(gAlrHist);
	AlarmsHistory();

END_ACTION
```

#### HMI.var - Local variables
```iecst
VAR
	AlarmsHistory : MpAlarmXHistory;
	AlarmsCore : MpAlarmXCore;
	xTest : BOOL;
	myValue : UDINT;
	xNone : BOOL;
	xActive : BOOL;
	xInactive : BOOL;
	xAck : BOOL;
	xUnAck : BOOL;
	myValue2 : DINT;
	myValueAck : DINT;
	xTest2 : BOOL;
	myValueAck2 : DINT;
	xSimulateMedia : BOOL;
	tonSimMedia : TON;
	dataInksHMI : REFERENCE TO stInks;
	iInkHMI : USINT := 1;
	strInkType : STRING[10];
	strPrintHeadType : STRING[10];
	iInkHMI_copy : USINT;
END_VAR
```

### Program Logical/InkBox/InkBoxCtrl/MainInkBox (IEC)

#### Variables.var
```iecst
VAR
	iIndex : USINT;
	iTemp1 : BOOL;
	dataInksInput : REFERENCE TO stInks;
	iCabinet : USINT;
	iInksInCabinet : USINT;
	iInkIndex : USINT;
	rPowerPerCabinet : REAL;
	rCabinetReductionTempPower : REAL;
	rMaxTempPower : REAL;
	rTotalInksInCabinet : REAL;
	xaExistingInks : ARRAY[0..MAX_LAST_INK] OF BOOL;
	xaExistingInksReseted : ARRAY[0..MAX_LAST_INK] OF BOOL;
	dataInksInParams : stInksParameters;
	CommandsReseted : InkboxCommands;
END_VAR
```

#### Cyclic.st
```iecst
PROGRAM _INIT

	VersionPLC;

	PLC_Init(ADR(gPLC));

	//Limit values for all possible Cabinets
	FOR iCabinet := 1 TO MAX_LAST_INK_CABINET DO
		gInkBox.Parameters.Cabinets[iCabinet].TotalInkSystems := MAX(2, gInkBox.Parameters.Cabinets[iCabinet].TotalInkSystems);
		gInkBox.Parameters.Cabinets[iCabinet].TotalInksPerPsu := MAX(1, gInkBox.Parameters.Cabinets[iCabinet].TotalInksPerPsu);
		gInkBox.Parameters.Cabinets[iCabinet].MaxTempPowerPsu := MAX(100, gInkBox.Parameters.Cabinets[iCabinet].MaxTempPowerPsu);
	END_FOR;

	FOR iIndex:=1 TO MAX_LAST_INK DO

		//Reference working data to the general data
		dataInksInput ACCESS ADR(gInks[iIndex]);

		IF dataInksInput.parSw.Config.iInkType <= 0 THEN
			dataInksInput.parSw.Config.iInkType:=lc_iInkMineral;
		END_IF
		IF dataInksInput.parSw.Config.iPrintHeadType <= 0 THEN
			dataInksInput.parSw.Config.iPrintHeadType:=lc_iPrintHeadSK1536;
		END_IF

		printHeadData_Nozomi2;

		dataInksInput.parameters.Temp.iBarsWithSamePsu := 1;

		dataInksInput.parSw.xEnabledBarToPrint := TRUE;

		dataInksInput.parSw.Config.iMappingBar := iIndex;

		dataInksInput.parSw.NegPump.rLowerLimMeniscusCritical := -120;
		dataInksInput.parSw.NegPump.rUpperLimMeniscusCritical := 70.0;

//		IF dataInksInput.parSw.PosPump.rSetPoint = 0 THEN
//			dataInksInput.parSw.PosPump.rSetPoint := 7.0;
//		END_IF
//		IF dataInksInput.parSw.NegPump.rSetPointMeniscus = 0 THEN
//			dataInksInput.parSw.NegPump.rSetPointMeniscus := 24;
//		END_IF
		IF dataInksInput.parSw.tiDripTime = 0 THEN
			dataInksInput.parSw.tiDripTime := MILLISECONDS_TO_TIME(300*iIndex);
		END_IF

		dataInksInput.signals.in.xPrintHeadsPsuOK := TRUE;

	END_FOR;

END_PROGRAM

PROGRAM _CYCLIC

	InternalPLC;

	//At least 1 cabinet
	gInkBox.Parameters.TotalCabinets := MAX(1, gInkBox.Parameters.TotalCabinets);

	FOR iCabinet := 1 TO MAX_LAST_INK_CABINET DO
		rTotalInksInCabinet := USINT_TO_REAL(gInkBox.Parameters.Cabinets[iCabinet].TotalInkSystems);
		rTotalInksInCabinet := 2 * brmceil(rTotalInksInCabinet/2);
		gInkBox.Parameters.Cabinets[iCabinet].TotalInkSystems := MAX(2, REAL_TO_USINT(rTotalInksInCabinet));

		gInkBox.Parameters.Cabinets[iCabinet].MaxTempPowerPsu := MAX(100, gInkBox.Parameters.Cabinets[iCabinet].MaxTempPowerPsu);

		gInkBox.Status.Cabinets[iCabinet].xExists := iCabinet <= gInkBox.Parameters.TotalCabinets;
	END_FOR

	iCabinet := 1;
	iInksInCabinet := 1;
	FOR iIndex:=1 TO MAX_LAST_INK DO

		//Reference working data to the general data
		dataInksInput ACCESS ADR(gInks[iIndex]);

		//If the bar system do not exist, assign an imposible mapping bar to consider uninstalled and remove alarms
		IF iIndex > gInkBox.Status.iTotalInks THEN
			dataInksInput.parSw.Config.iMappingBar := -1;
		ELSE
			dataInksInput.parSw.Config.iMappingBar := iIndex;
		END_IF

		IF dataInksInput.parSw.Config.iInkType <= 0 THEN
			dataInksInput.parSw.Config.iInkType:=lc_iInkMineral;
		END_IF
		IF dataInksInput.parSw.Config.iPrintHeadType <= 0 THEN
			dataInksInput.parSw.Config.iPrintHeadType:=lc_iPrintHeadSK1536;
		END_IF

		//Assign current data to working data
		dataInksInParams := dataInksInput.parameters;

		printHeadData;

		//Assign working data to Ink parameters
		dataInksInput.parameters := dataInksInParams;

		dataInksInput.parameters.Temp.iBarsWithSameBlock := gInkBox.Parameters.Cabinets[iCabinet].TotalInkSystems;
		dataInksInput.parameters.Temp.iBarsWithSamePsu := gInkBox.Parameters.Cabinets[iCabinet].TotalInksPerPsu;

		dataInksInput.commands.xErrorRst := gInkBox.Commands.xReset;
		dataInksInput.commands.xMute := gInkBox.Commands.xMute;

		//Go to next Ink System
		iInksInCabinet := iInksInCabinet + 1;
		IF iInksInCabinet > gInkBox.Parameters.Cabinets[iCabinet].TotalInkSystems THEN
			iInksInCabinet := 1;
			iCabinet := iCabinet + 1;
		END_IF

	END_FOR

	//Calculate Power per Cabinet
	iInkIndex := 1; //Incremented just in existing cabinets
	xaExistingInks := xaExistingInksReseted;
	FOR iCabinet := 1 TO MAX_LAST_INK_CABINET DO
		CalculatePowerPerCabinet;
	END_FOR
	gInkBox.Status.iTotalInks := iInkIndex -1;
	gInkBox.Status.ExistingInks := xaExistingInks;

	//Limit total InksSystems to 12

	//Assign max data to each InkSystem
	iInkIndex := 1;
	FOR iCabinet := 1 TO MAX_LAST_INK_CABINET DO
		AssignPowerPerCabinet;
	END_FOR

	gInkBox.Commands := CommandsReseted;

END_PROGRAM
```

#### VersionPLC.st
```iecst
ACTION VersionPLC:

	// Version
	gPLC.iVersion0:= 1;	// Major version
	gPLC.iVersion1:= 3;	// Refactoring
	gPLC.iVersion2:= 225;	// Updated ExtPack
	gPLC.iVersion3:= 32;	// Version

END_ACTION
```

### Program Logical/InkBox/PhysicalMapping/PhysicalMapInputs (IEC)

#### InputsInkBox.st - PhysicalInputs
```iecst
ACTION InputsInkBox:

	// GROUP _10x
	gInks[1].signals.in.xPrintHeadsPsuOK := NOT X20DIF371_101.DInput[1];
	gInks[1].signals.in.xKlixonTriggered := X20DIF371_101.DInput[3];
	gInks[1].signals.in.xOverpressure := NOT X20DIF371_101.DInput[5];
	gInks[1].signals.in.xMaxLevel := X20DIF371_101.DInput[7];
	gInks[1].signals.in.xMinLevel := X20DIF371_101.DInput[9];

	gInks[2].signals.in.xPrintHeadsPsuOK := NOT X20DIF371_101.DInput[2];
	gInks[2].signals.in.xKlixonTriggered := X20DIF371_101.DInput[4];
	gInks[2].signals.in.xOverpressure := NOT X20DIF371_101.DInput[6];
	gInks[2].signals.in.xMaxLevel := X20DIF371_101.DInput[8];
	gInks[2].signals.in.xMinLevel := X20DIF371_101.DInput[10];

	gInks[1].signals.in.iVacuum1Raw := X20AI4322_102.AInput[1];
	gInks[1].signals.in.xVacuum1SensorError := StatusAnalogInputBroken( X20AI4322_102.ModuleOk, X20AI4322_102.Status01, X20AI4322_102.Status02, 1);
	gInks[1].signals.in.iVacuum2Raw := X20AI4322_102.AInput[3];
	gInks[1].signals.in.xVacuum2SensorError := StatusAnalogInputBroken( X20AI4322_102.ModuleOk, X20AI4322_102.Status01, X20AI4322_102.Status02, 3);

	gInks[2].signals.in.iVacuum1Raw := X20AI4322_102.AInput[2];
	gInks[2].signals.in.xVacuum1SensorError := StatusAnalogInputBroken( X20AI4322_102.ModuleOk, X20AI4322_102.Status01, X20AI4322_102.Status02, 2);
	gInks[2].signals.in.iVacuum2Raw := X20AI4322_102.AInput[4];
	gInks[2].signals.in.xVacuum2SensorError := StatusAnalogInputBroken( X20AI4322_102.ModuleOk, X20AI4322_102.Status01, X20AI4322_102.Status02, 4);

	gInks[1].signals.in.iTemperatureRaw := X20AT2222_103.TempInput[1];
	gInks[1].signals.in.xTempSensorError := StatusTemperatureInput(X20AT2222_103.Status01, 1);
	gInks[1].signals.in.iTemperatureTankRaw := X20AT2222_103.TempInput[3];
	gInks[1].signals.in.xTempTankSensorError := StatusTemperatureInput(X20AT2222_103.Status01, 3);

	gInks[2].signals.in.iTemperatureRaw := X20AT2222_103.TempInput[2];
	gInks[2].signals.in.xTempSensorError := StatusTemperatureInput(X20AT2222_103.Status01, 2);
	gInks[2].signals.in.iTemperatureTankRaw := X20AT2222_103.TempInput[4];
	gInks[2].signals.in.xTempTankSensorError := StatusTemperatureInput(X20AT2222_103.Status01, 4);

	// GROUP _20x
	gInks[3].signals.in.xPrintHeadsPsuOK := NOT X20DIF371_201.DInput[1];
	gInks[3].signals.in.xKlixonTriggered := X20DIF371_201.DInput[3];
	gInks[3].signals.in.xOverpressure := NOT X20DIF371_201.DInput[5];
	gInks[3].signals.in.xMaxLevel := X20DIF371_201.DInput[7];
	gInks[3].signals.in.xMinLevel := X20DIF371_201.DInput[9];

	gInks[4].signals.in.xPrintHeadsPsuOK := NOT X20DIF371_201.DInput[2];
	gInks[4].signals.in.xKlixonTriggered := X20DIF371_201.DInput[4];
	gInks[4].signals.in.xOverpressure := NOT X20DIF371_201.DInput[6];
	gInks[4].signals.in.xMaxLevel := X20DIF371_201.DInput[8];
	gInks[4].signals.in.xMinLevel := X20DIF371_201.DInput[10];

	gInks[3].signals.in.iVacuum1Raw := X20AI4322_202.AInput[1];
	gInks[3].signals.in.xVacuum1SensorError := StatusAnalogInputBroken( X20AI4322_202.ModuleOk, X20AI4322_202.Status01, X20AI4322_202.Status02, 1);
	gInks[3].signals.in.iVacuum2Raw := X20AI4322_202.AInput[3];
	gInks[3].signals.in.xVacuum2SensorError := StatusAnalogInputBroken( X20AI4322_202.ModuleOk, X20AI4322_202.Status01, X20AI4322_202.Status02, 3);

	gInks[4].signals.in.iVacuum1Raw := X20AI4322_202.AInput[2];
	gInks[4].signals.in.xVacuum1SensorError := StatusAnalogInputBroken( X20AI4322_202.ModuleOk, X20AI4322_202.Status01, X20AI4322_202.Status02, 2);
	gInks[4].signals.in.iVacuum2Raw := X20AI4322_202.AInput[4];
	gInks[4].signals.in.xVacuum2SensorError := StatusAnalogInputBroken( X20AI4322_202.ModuleOk, X20AI4322_202.Status01, X20AI4322_202.Status02, 4);

	gInks[3].signals.in.iTemperatureRaw := X20AT2222_203.TempInput[1];
	gInks[3].signals.in.xTempSensorError := StatusTemperatureInput(X20AT2222_203.Status01, 1);
	gInks[3].signals.in.iTemperatureTankRaw := X20AT2222_203.TempInput[3];
	gInks[3].signals.in.xTempTankSensorError := StatusTemperatureInput(X20AT2222_203.Status01, 3);

	gInks[4].signals.in.iTemperatureRaw := X20AT2222_203.TempInput[2];
	gInks[4].signals.in.xTempSensorError := StatusTemperatureInput(X20AT2222_203.Status01, 2);
	gInks[4].signals.in.iTemperatureTankRaw := X20AT2222_203.TempInput[4];
	gInks[4].signals.in.xTempTankSensorError := StatusTemperatureInput(X20AT2222_203.Status01, 4);

	// GROUP _30x
	gInks[5].signals.in.xPrintHeadsPsuOK := NOT X20DIF371_301.DInput[1];
	gInks[5].signals.in.xKlixonTriggered := X20DIF371_301.DInput[3];
	gInks[5].signals.in.xOverpressure := NOT X20DIF371_301.DInput[5];
	gInks[5].signals.in.xMaxLevel := X20DIF371_301.DInput[7];
	gInks[5].signals.in.xMinLevel := X20DIF371_301.DInput[9];

	gInks[6].signals.in.xPrintHeadsPsuOK := NOT X20DIF371_301.DInput[2];
	gInks[6].signals.in.xKlixonTriggered := X20DIF371_301.DInput[4];
	gInks[6].signals.in.xOverpressure := NOT X20DIF371_301.DInput[6];
	gInks[6].signals.in.xMaxLevel := X20DIF371_301.DInput[8];
	gInks[6].signals.in.xMinLevel := X20DIF371_301.DInput[10];

	gInks[5].signals.in.iVacuum1Raw := X20AI4322_302.DInput[1];
	gInks[5].signals.in.xVacuum1SensorError := StatusAnalogInputBroken( X20AI4322_302.ModuleOk, X20AI4322_302.Status01, X20AI4322_302.Status02, 1);
	gInks[5].signals.in.iVacuum2Raw := X20AI4322_302.DInput[3];
	gInks[5].signals.in.xVacuum2SensorError := StatusAnalogInputBroken( X20AI4322_302.ModuleOk, X20AI4322_302.Status01, X20AI4322_302.Status02, 3);

	gInks[6].signals.in.iVacuum1Raw := X20AI4322_302.DInput[2];
	gInks[6].signals.in.xVacuum1SensorError := StatusAnalogInputBroken( X20AI4322_302.ModuleOk, X20AI4322_302.Status01, X20AI4322_302.Status02, 2);
	gInks[6].signals.in.iVacuum2Raw := X20AI4322_302.DInput[4];
	gInks[6].signals.in.xVacuum2SensorError := StatusAnalogInputBroken( X20AI4322_302.ModuleOk, X20AI4322_302.Status01, X20AI4322_302.Status02, 4);

	gInks[5].signals.in.iTemperatureRaw := X20AT2222_303.TempInput[1];
	gInks[5].signals.in.xTempSensorError := StatusTemperatureInput(X20AT2222_303.Status01, 1);
	gInks[5].signals.in.iTemperatureTankRaw := X20AT2222_303.TempInput[3];
	gInks[5].signals.in.xTempTankSensorError := StatusTemperatureInput(X20AT2222_303.Status01, 3);

	gInks[6].signals.in.iTemperatureRaw := X20AT2222_303.TempInput[2];
	gInks[6].signals.in.xTempSensorError := StatusTemperatureInput(X20AT2222_303.Status01, 2);
	gInks[6].signals.in.iTemperatureTankRaw := X20AT2222_303.TempInput[4];
	gInks[6].signals.in.xTempTankSensorError := StatusTemperatureInput(X20AT2222_303.Status01, 4);

END_ACTION
```

### Program Logical/InkBox/PhysicalMapping/PhysicalMapOutputs

#### PhysicalMapOutputs.var
```iecst
VAR
	iIndexInksSlow : USINT;
	iIndexPhysicalInksSlow : USINT;
	inksOutputsReseted : stInksSignalsOut;
END_VAR
```

#### MappingOutputs.st
```iecst
PROGRAM _CYCLIC

	//If in automation runtime, do not assign physical mapping
	IF gMachine.St.HwData.Family = FAMILY_BRAUTOMATIONRUNTIME THEN
		RETURN;
	END_IF

	OutputsInkBox;

	// ####################################################################
	// ####################################################################
	//  Reset bar outputs if do not have any logical bar mapped
	// ####################################################################

	// Reset the index if the index is not valid
	IF iIndexPhysicalInksSlow = 0 OR iIndexPhysicalInksSlow > MAX_LAST_INK THEN
		//Resetart index
		iIndexPhysicalInksSlow := 1;
		iIndexInksSlow := 1;
	END_IF
	IF iIndexInksSlow = 0 OR iIndexInksSlow > MAX_LAST_INK THEN iIndexInksSlow := 1; END_IF

	//If the physical bar has a logical bar in that position, go to next physical bar and reset logical index bar
	IF iIndexPhysicalInksSlow = gInks[iIndexInksSlow].parSw.Config.iMappingBar THEN
		iIndexPhysicalInksSlow := iIndexPhysicalInksSlow + 1;
		iIndexInksSlow := 1;
	ELSE
		iIndexInksSlow := iIndexInksSlow + 1;
	END_IF

	//If there is no logical bar with the mapping of the physical position, reset the outputs
	IF iIndexInksSlow > MAX_LAST_INK THEN

		//Reset the outputs to avoid keeping the outputs active
		gInksOutputs[iIndexPhysicalInksSlow] := inksOutputsReseted;

		//Go to next physical and reset logical index bar
		iIndexPhysicalInksSlow := iIndexPhysicalInksSlow + 1;
		iIndexInksSlow := 1;
	END_IF

END_PROGRAM
```

- PrintJig_v10.7z (binary file, 1195662 bytes)
- Program Logical/InkBox/Transport/Transport (IEC) (no source held here)

### Package Logical/AsSafetySolution - AsSafety design sample

- Visualisation Logical/AsSafetySolution/Panel (not shown)

### Library Logical/AsSafetySolution/SafetySample
